(****************************** 10-001-0215-00-0 ************************************)
(*************************** ProBoxElement with one Motor *******************************)
// Configuration element 
fbEL_10_001_0215_00_0.ConfigElement.ElementName                     := '10-001-0215-00-0'; // Element name 
fbEL_10_001_0215_00_0.ConfigElement.eElementNumber                  := E_10_001_0215_00_0; // Number of the element 
fbEL_10_001_0215_00_0.ConfigElement.eSlaveElementNumber_34          := E_ElementNumber.E_BEGIN_ELEMENT; // Link from Master to slave element
fbEL_10_001_0215_00_0.ConfigElement.eElementType                    := E_ElementType.NO_TYPE; // No specific type

// Register element 
ElementRegistry[E_10_001_0215_00_0].Enable                          := TRUE; // Object is called
ElementRegistry[E_10_001_0215_00_0].eElementNumber                  := fbEL_10_001_0215_00_0.ConfigElement.eElementNumber; 

(****************************** 10-001-0215-01-0 ************************************)
(************************** ProBox Straight Transport *******************************)
// Configuration function
fbF_10_001_0215_01_0.ConfigFunction.FunctionName                       := '10-001-0215-01-0'; // Function name
fbF_10_001_0215_01_0.ConfigFunction.eFunctionNumber                    := F_10_001_0215_01_0; // Number of the function
fbF_10_001_0215_01_0.ConfigFunction.eElementLink                       := E_ElementNumber.E_10_001_0215_00_0;
fbF_10_001_0215_01_0.ConfigFunction.FunctionLink.eFunctionNumber       := E_FunctionNumber.F_BEGIN_FUNCTION;
fbF_10_001_0215_01_0.ConfigFunction.FunctionLink.ZoneNumber            := 0;
fbF_10_001_0215_01_0.ConfigFunction.eAdjacentFunctionNumberSide[1]     := E_FunctionNumber.F_10_001_0214_01_0;
fbF_10_001_0215_01_0.ConfigFunction.eAdjacentFunctionNumberSide[2]     := E_FunctionNumber.F_10_001_0215_02_0;
fbF_10_001_0215_01_0.ConfigFunction.ePrevFunctionNumber                := E_FunctionNumber.F_10_001_0214_01_0;
fbF_10_001_0215_01_0.ConfigFunction.eNextFunctionNumber                := E_FunctionNumber.F_10_001_0215_02_0;
fbF_10_001_0215_01_0.ConfigFunction.NumberOfZones                      := 1;
//Config zone 1
fbF_10_001_0215_01_0.ConfigFunction.Zone[1].ZoneName                   := '10-001-0215-01-1';
fbF_10_001_0215_01_0.ConfigFunction.Zone[1].EnableMFC                  := TRUE;
fbF_10_001_0215_01_0.ConfigFunction.Zone[1].EnableSimultaneousTransport:= FALSE; //Disable Simultaneous transport for multi zone functions
fbF_10_001_0215_01_0.ConfigFunction.Zone[1].EnableLatchOccupiedState   := TRUE;
fbF_10_001_0215_01_0.ConfigFunction.Zone[1].Length[1]                  := INT_TO_UINT(2600 / fbF_10_001_0215_01_0.ConfigFunction.NumberOfZones);	//Zone length (ie element length / number of zones)

// Register function
FunctionRegistry[F_10_001_0215_01_0].Enable                            := TRUE; (* Function will be called *)
FunctionRegistry[F_10_001_0215_01_0].eFunctionNumber                   := fbF_10_001_0215_01_0.ConfigFunction.eFunctionNumber; // Registration number


(****************************** 10-001-0215-02-0 ************************************)
(************************** ProBox Straight Transport *******************************)
// Configuration function
fbF_10_001_0215_02_0.ConfigFunction.FunctionName                       := '10-001-0215-02-0'; // Function name
fbF_10_001_0215_02_0.ConfigFunction.eFunctionNumber                    := F_10_001_0215_02_0; // Number of the function
fbF_10_001_0215_02_0.ConfigFunction.eElementLink                       := E_ElementNumber.E_10_001_0215_00_0;
fbF_10_001_0215_02_0.ConfigFunction.FunctionLink.eFunctionNumber       := E_FunctionNumber.F_BEGIN_FUNCTION;
fbF_10_001_0215_02_0.ConfigFunction.FunctionLink.ZoneNumber            := 0;
fbF_10_001_0215_02_0.ConfigFunction.eAdjacentFunctionNumberSide[1]     := E_FunctionNumber.F_10_001_0215_01_0;
fbF_10_001_0215_02_0.ConfigFunction.eAdjacentFunctionNumberSide[2]     := E_FunctionNumber.F_BEGIN_FUNCTION;
fbF_10_001_0215_02_0.ConfigFunction.ePrevFunctionNumber                := E_FunctionNumber.F_10_001_0215_01_0;
fbF_10_001_0215_02_0.ConfigFunction.eNextFunctionNumber                := E_FunctionNumber.F_BEGIN_FUNCTION;
fbF_10_001_0215_02_0.ConfigFunction.NumberOfZones                      := 1;
//Config zone 1
fbF_10_001_0215_02_0.ConfigFunction.Zone[1].ZoneName                   := '10-001-0215-02-1';
fbF_10_001_0215_02_0.ConfigFunction.Zone[1].EnableMFC                  := TRUE;
fbF_10_001_0215_02_0.ConfigFunction.Zone[1].EnableSimultaneousTransport:= FALSE; //Disable Simultaneous transport for multi zone functions
fbF_10_001_0215_02_0.ConfigFunction.Zone[1].EnableLatchOccupiedState   := TRUE;
fbF_10_001_0215_02_0.ConfigFunction.Zone[1].Length[1]                  := INT_TO_UINT(2600 / fbF_10_001_0215_02_0.ConfigFunction.NumberOfZones);	//Zone length (ie element length / number of zones)

// Register function
FunctionRegistry[F_10_001_0215_02_0].Enable                            := TRUE; (* Function will be called *)
FunctionRegistry[F_10_001_0215_02_0].eFunctionNumber                   := fbF_10_001_0215_02_0.ConfigFunction.eFunctionNumber; // Registration number


(****************************** 10-001-0215-03-0 ************************************)
(******************************* Crane Handover/Takeover ***********************************)
// Configuration function 
fbF_10_001_0215_03_0.ConfigFunction.FunctionName                      	 := '10-001-0215-03-0'; (* Function name *)
fbF_10_001_0215_03_0.ConfigFunction.eFunctionNumber                  	 := F_10_001_0215_03_0; (* Number of the function *)
fbF_10_001_0215_03_0.ConfigFunction.eElementLink                     	 := E_ElementNumber.E_10_001_0215_00_0; 
fbF_10_001_0215_03_0.ConfigFunction.FunctionLink.eFunctionNumber     	 := E_FunctionNumber.F_10_001_0215_01_0;	//Addon link to function, this is auto generated, an may need to be changed.
fbF_10_001_0215_03_0.ConfigFunction.FunctionLink.ZoneNumber         	 := 1;		

fbF_10_001_0215_03_0.Config.TimeoutValueLift							 := T#10S;								// Timeout value for lifting
fbF_10_001_0215_03_0.Config.HomePosFree								 := E_Positions_LiftControl.DOWN;		// Homeposition lift when zone free
fbF_10_001_0215_03_0.Config.HomePosOccupied							 := E_Positions_LiftControl.UP;			// Homeposition lift when zone occupied
fbF_10_001_0215_03_0.Config.CraneXoverType								 := E_CvCraneXoverType.eCOMBINATION; 	// Function Crane Deposit and Crane Pickup
fbF_10_001_0215_03_0.Config.LiftEnabled								 := FALSE;								// config if station has lift	
fbF_10_001_0215_03_0.Config.CfgMotorTransfer.EnableMotorTransferTU		 := FALSE;  								// Enable or Disable motor drive chain transfer 
fbF_10_001_0215_03_0.Config.CfgMotorTransfer.HandoverMotorDir			 := E_DriveDirection.FWD; 				// Direction during handover
fbF_10_001_0215_03_0.Config.CfgMotorTransfer.TakeoverMotorDir			 := E_DriveDirection.FWD; 				// Direction during takeover
fbF_10_001_0215_03_0.Config.CfgMotorTransfer.MotorDriveTimeout			 := T#20S;	
fbF_10_001_0215_03_0.Config.CfgMotorTransfer.MotorSpeed				 := E_ProBoxMotorSpeed.NORMAL;

fbF_10_001_0215_03_0.Config.CraneCom.TCP_IP_Config.ChannelName          := 'CraneTCPIPcom';
fbF_10_001_0215_03_0.Config.CraneCom.TCP_IP_Config.EnableConnection     := TRUE;
fbF_10_001_0215_03_0.Config.CraneCom.TCP_IP_Config.RemoteHost           := '192.168.1.1';
fbF_10_001_0215_03_0.Config.CraneCom.TCP_IP_Config.RemotePort           := 2011;
fbF_10_001_0215_03_0.Config.CraneCom.TCP_IP_Config.LocalHost            := '0.0.0.0';
fbF_10_001_0215_03_0.Config.CraneCom.TCP_IP_Config.LocalPort            := 5001;
fbF_10_001_0215_03_0.Config.CraneCom.TCP_IP_Config.Server               := FALSE;
fbF_10_001_0215_03_0.Config.CraneCom.TCP_IP_Config.ConnectTimeout       := T#10S;
fbF_10_001_0215_03_0.Config.CraneCom.TCP_IP_Config.ClientRetryInterval  := T#5S;
fbF_10_001_0215_03_0.Config.CraneCom.TCP_IP_Config.ServerRetryInterval  := T#1S;
fbF_10_001_0215_03_0.Config.CraneCom.TCP_IP_Config.AcceptPollInterval   := T#10S;
fbF_10_001_0215_03_0.Config.CraneCom.TCP_IP_Config.EnableDebugMsg       := TRUE;	


// Register function 
FunctionRegistry[F_10_001_0215_03_0].Enable                          	 := TRUE; (* Function will be called *)
FunctionRegistry[F_10_001_0215_03_0].eFunctionNumber                  	 := fbF_10_001_0215_03_0.ConfigFunction.eFunctionNumber; (* Registration number *)


(****************************** 10-001-0216-00-0 ************************************)
(*************************** ProBoxElement with one Motor *******************************)
// Configuration element 
fbEL_10_001_0216_00_0.ConfigElement.ElementName                     := '10-001-0216-00-0'; // Element name 
fbEL_10_001_0216_00_0.ConfigElement.eElementNumber                  := E_10_001_0216_00_0; // Number of the element 
fbEL_10_001_0216_00_0.ConfigElement.eSlaveElementNumber_34          := E_ElementNumber.E_BEGIN_ELEMENT; // Link from Master to slave element
fbEL_10_001_0216_00_0.ConfigElement.eElementType                    := E_ElementType.NO_TYPE; // No specific type

// Register element 
ElementRegistry[E_10_001_0216_00_0].Enable                          := TRUE; // Object is called
ElementRegistry[E_10_001_0216_00_0].eElementNumber                  := fbEL_10_001_0216_00_0.ConfigElement.eElementNumber; 

(****************************** 10-001-0216-01-0 ************************************)
(************************** ProBox Straight Transport *******************************)
// Configuration function
fbF_10_001_0216_01_0.ConfigFunction.FunctionName                       := '10-001-0216-01-0'; // Function name
fbF_10_001_0216_01_0.ConfigFunction.eFunctionNumber                    := F_10_001_0216_01_0; // Number of the function
fbF_10_001_0216_01_0.ConfigFunction.eElementLink                       := E_ElementNumber.E_10_001_0216_00_0;
fbF_10_001_0216_01_0.ConfigFunction.FunctionLink.eFunctionNumber       := E_FunctionNumber.F_BEGIN_FUNCTION;
fbF_10_001_0216_01_0.ConfigFunction.FunctionLink.ZoneNumber            := 0;
fbF_10_001_0216_01_0.ConfigFunction.eAdjacentFunctionNumberSide[1]     := E_FunctionNumber.F_BEGIN_FUNCTION;
fbF_10_001_0216_01_0.ConfigFunction.eAdjacentFunctionNumberSide[2]     := E_FunctionNumber.F_10_001_0217_01_0;
fbF_10_001_0216_01_0.ConfigFunction.ePrevFunctionNumber                := E_FunctionNumber.F_BEGIN_FUNCTION;
fbF_10_001_0216_01_0.ConfigFunction.eNextFunctionNumber                := E_FunctionNumber.F_10_001_0217_01_0;
fbF_10_001_0216_01_0.ConfigFunction.NumberOfZones                      := 2;
//Config zone 1
fbF_10_001_0216_01_0.ConfigFunction.Zone[1].ZoneName                   := '10-001-0216-01-1';
fbF_10_001_0216_01_0.ConfigFunction.Zone[1].EnableMFC                  := TRUE;
fbF_10_001_0216_01_0.ConfigFunction.Zone[1].EnableSimultaneousTransport:= TRUE; //Enable Simultaneous transport for multi zone functions
fbF_10_001_0216_01_0.ConfigFunction.Zone[1].EnableLatchOccupiedState   := TRUE;
fbF_10_001_0216_01_0.ConfigFunction.Zone[1].Length[1]                  := INT_TO_UINT(2600 / fbF_10_001_0216_01_0.ConfigFunction.NumberOfZones);	//Zone length (ie element length / number of zones)

//Config remaining zones equal to zone 1.
fbF_10_001_0216_01_0.ConfigFunction.Zone[2]                            := fbF_10_001_0216_01_0.ConfigFunction.Zone[1];
fbF_10_001_0216_01_0.ConfigFunction.Zone[2].ZoneName                   := '10-001-0216-01-2';

fbF_10_001_0216_01_0.Config.TwoSensorFunction                          := FALSE; // Slugging sensor present

// Register function
FunctionRegistry[F_10_001_0216_01_0].Enable                            := TRUE; (* Function will be called *)
FunctionRegistry[F_10_001_0216_01_0].eFunctionNumber                   := fbF_10_001_0216_01_0.ConfigFunction.eFunctionNumber; // Registration number


(****************************** 10-001-0216-02-0 ************************************)
(******************************* Crane Handover/Takeover ***********************************)
// Configuration function 
fbF_10_001_0216_02_0.ConfigFunction.FunctionName                      	 := '10-001-0216-02-0'; (* Function name *)
fbF_10_001_0216_02_0.ConfigFunction.eFunctionNumber                  	 := F_10_001_0216_02_0; (* Number of the function *)
fbF_10_001_0216_02_0.ConfigFunction.eElementLink                     	 := E_ElementNumber.E_10_001_0216_00_0; 
fbF_10_001_0216_02_0.ConfigFunction.FunctionLink.eFunctionNumber     	 := E_FunctionNumber.F_10_001_0216_01_0;	//Addon link to function, this is auto generated, an may need to be changed.
fbF_10_001_0216_02_0.ConfigFunction.FunctionLink.ZoneNumber         	 := 1;		

fbF_10_001_0216_02_0.Config.TimeoutValueLift							 := T#10S;								// Timeout value for lifting
fbF_10_001_0216_02_0.Config.HomePosFree								 := E_Positions_LiftControl.DOWN;		// Homeposition lift when zone free
fbF_10_001_0216_02_0.Config.HomePosOccupied							 := E_Positions_LiftControl.UP;			// Homeposition lift when zone occupied
fbF_10_001_0216_02_0.Config.CraneXoverType								 := E_CvCraneXoverType.eCOMBINATION; 	// Function Crane Deposit and Crane Pickup
fbF_10_001_0216_02_0.Config.LiftEnabled								 := FALSE;								// config if station has lift	
fbF_10_001_0216_02_0.Config.CfgMotorTransfer.EnableMotorTransferTU		 := FALSE;  								// Enable or Disable motor drive chain transfer 
fbF_10_001_0216_02_0.Config.CfgMotorTransfer.HandoverMotorDir			 := E_DriveDirection.FWD; 				// Direction during handover
fbF_10_001_0216_02_0.Config.CfgMotorTransfer.TakeoverMotorDir			 := E_DriveDirection.FWD; 				// Direction during takeover
fbF_10_001_0216_02_0.Config.CfgMotorTransfer.MotorDriveTimeout			 := T#20S;	
fbF_10_001_0216_02_0.Config.CfgMotorTransfer.MotorSpeed				 := E_ProBoxMotorSpeed.NORMAL;

fbF_10_001_0216_02_0.Config.CraneCom.TCP_IP_Config.ChannelName          := 'CraneTCPIPcom';
fbF_10_001_0216_02_0.Config.CraneCom.TCP_IP_Config.EnableConnection     := TRUE;
fbF_10_001_0216_02_0.Config.CraneCom.TCP_IP_Config.RemoteHost           := '192.168.1.1';
fbF_10_001_0216_02_0.Config.CraneCom.TCP_IP_Config.RemotePort           := 2011;
fbF_10_001_0216_02_0.Config.CraneCom.TCP_IP_Config.LocalHost            := '0.0.0.0';
fbF_10_001_0216_02_0.Config.CraneCom.TCP_IP_Config.LocalPort            := 5001;
fbF_10_001_0216_02_0.Config.CraneCom.TCP_IP_Config.Server               := FALSE;
fbF_10_001_0216_02_0.Config.CraneCom.TCP_IP_Config.ConnectTimeout       := T#10S;
fbF_10_001_0216_02_0.Config.CraneCom.TCP_IP_Config.ClientRetryInterval  := T#5S;
fbF_10_001_0216_02_0.Config.CraneCom.TCP_IP_Config.ServerRetryInterval  := T#1S;
fbF_10_001_0216_02_0.Config.CraneCom.TCP_IP_Config.AcceptPollInterval   := T#10S;
fbF_10_001_0216_02_0.Config.CraneCom.TCP_IP_Config.EnableDebugMsg       := TRUE;	


// Register function 
FunctionRegistry[F_10_001_0216_02_0].Enable                          	 := TRUE; (* Function will be called *)
FunctionRegistry[F_10_001_0216_02_0].eFunctionNumber                  	 := fbF_10_001_0216_02_0.ConfigFunction.eFunctionNumber; (* Registration number *)


(****************************** 10-001-0217-00-0 ************************************)
(*************************** ProBoxElement with one Motor *******************************)
// Configuration element 
fbEL_10_001_0217_00_0.ConfigElement.ElementName                     := '10-001-0217-00-0'; // Element name 
fbEL_10_001_0217_00_0.ConfigElement.eElementNumber                  := E_10_001_0217_00_0; // Number of the element 
fbEL_10_001_0217_00_0.ConfigElement.eSlaveElementNumber_34          := E_ElementNumber.E_BEGIN_ELEMENT; // Link from Master to slave element
fbEL_10_001_0217_00_0.ConfigElement.eElementType                    := E_ElementType.NO_TYPE; // No specific type

// Register element 
ElementRegistry[E_10_001_0217_00_0].Enable                          := TRUE; // Object is called
ElementRegistry[E_10_001_0217_00_0].eElementNumber                  := fbEL_10_001_0217_00_0.ConfigElement.eElementNumber; 

(****************************** 10-001-0217-01-0 ************************************)
(************************** ProBox Straight Transport *******************************)
// Configuration function
fbF_10_001_0217_01_0.ConfigFunction.FunctionName                       := '10-001-0217-01-0'; // Function name
fbF_10_001_0217_01_0.ConfigFunction.eFunctionNumber                    := F_10_001_0217_01_0; // Number of the function
fbF_10_001_0217_01_0.ConfigFunction.eElementLink                       := E_ElementNumber.E_10_001_0217_00_0;
fbF_10_001_0217_01_0.ConfigFunction.FunctionLink.eFunctionNumber       := E_FunctionNumber.F_BEGIN_FUNCTION;
fbF_10_001_0217_01_0.ConfigFunction.FunctionLink.ZoneNumber            := 0;
fbF_10_001_0217_01_0.ConfigFunction.eAdjacentFunctionNumberSide[1]     := E_FunctionNumber.F_10_001_0216_01_0;
fbF_10_001_0217_01_0.ConfigFunction.eAdjacentFunctionNumberSide[2]     := E_FunctionNumber.F_10_001_0212_01_0;
fbF_10_001_0217_01_0.ConfigFunction.ePrevFunctionNumber                := E_FunctionNumber.F_10_001_0216_01_0;
fbF_10_001_0217_01_0.ConfigFunction.eNextFunctionNumber                := E_FunctionNumber.F_10_001_0212_01_0;
fbF_10_001_0217_01_0.ConfigFunction.NumberOfZones                      := 1;
//Config zone 1
fbF_10_001_0217_01_0.ConfigFunction.Zone[1].ZoneName                   := '10-001-0217-01-1';
fbF_10_001_0217_01_0.ConfigFunction.Zone[1].EnableMFC                  := TRUE;
fbF_10_001_0217_01_0.ConfigFunction.Zone[1].EnableSimultaneousTransport:= FALSE; //Disable Simultaneous transport for multi zone functions
fbF_10_001_0217_01_0.ConfigFunction.Zone[1].EnableLatchOccupiedState   := TRUE;
fbF_10_001_0217_01_0.ConfigFunction.Zone[1].Length[1]                  := INT_TO_UINT(3000 / fbF_10_001_0217_01_0.ConfigFunction.NumberOfZones);	//Zone length (ie element length / number of zones)

// Register function
FunctionRegistry[F_10_001_0217_01_0].Enable                            := TRUE; (* Function will be called *)
FunctionRegistry[F_10_001_0217_01_0].eFunctionNumber                   := fbF_10_001_0217_01_0.ConfigFunction.eFunctionNumber; // Registration number


(****************************** 10-001-0218-00-0 ************************************)
(*************************** ProBoxElement with one Motor *******************************)
// Configuration element 
fbEL_10_001_0218_00_0.ConfigElement.ElementName                     := '10-001-0218-00-0'; // Element name 
fbEL_10_001_0218_00_0.ConfigElement.eElementNumber                  := E_10_001_0218_00_0; // Number of the element 
fbEL_10_001_0218_00_0.ConfigElement.eSlaveElementNumber_34          := E_ElementNumber.E_BEGIN_ELEMENT; // Link from Master to slave element
fbEL_10_001_0218_00_0.ConfigElement.eElementType                    := E_ElementType.NO_TYPE; // No specific type

// Register element 
ElementRegistry[E_10_001_0218_00_0].Enable                          := TRUE; // Object is called
ElementRegistry[E_10_001_0218_00_0].eElementNumber                  := fbEL_10_001_0218_00_0.ConfigElement.eElementNumber; 

(****************************** 10-001-0218-01-0 ************************************)
(************************** ProBox Straight Transport *******************************)
// Configuration function
fbF_10_001_0218_01_0.ConfigFunction.FunctionName                       := '10-001-0218-01-0'; // Function name
fbF_10_001_0218_01_0.ConfigFunction.eFunctionNumber                    := F_10_001_0218_01_0; // Number of the function
fbF_10_001_0218_01_0.ConfigFunction.eElementLink                       := E_ElementNumber.E_10_001_0218_00_0;
fbF_10_001_0218_01_0.ConfigFunction.FunctionLink.eFunctionNumber       := E_FunctionNumber.F_BEGIN_FUNCTION;
fbF_10_001_0218_01_0.ConfigFunction.FunctionLink.ZoneNumber            := 0;
fbF_10_001_0218_01_0.ConfigFunction.eAdjacentFunctionNumberSide[1]     := E_FunctionNumber.F_10_001_0212_01_0;
fbF_10_001_0218_01_0.ConfigFunction.eAdjacentFunctionNumberSide[2]     := E_FunctionNumber.F_10_001_0219_01_0;
fbF_10_001_0218_01_0.ConfigFunction.ePrevFunctionNumber                := E_FunctionNumber.F_10_001_0212_01_0;
fbF_10_001_0218_01_0.ConfigFunction.eNextFunctionNumber                := E_FunctionNumber.F_10_001_0219_01_0;
fbF_10_001_0218_01_0.ConfigFunction.NumberOfZones                      := 2;
//Config zone 1
fbF_10_001_0218_01_0.ConfigFunction.Zone[1].ZoneName                   := '10-001-0218-01-1';
fbF_10_001_0218_01_0.ConfigFunction.Zone[1].EnableMFC                  := TRUE;
fbF_10_001_0218_01_0.ConfigFunction.Zone[1].EnableSimultaneousTransport:= TRUE; //Enable Simultaneous transport for multi zone functions
fbF_10_001_0218_01_0.ConfigFunction.Zone[1].EnableLatchOccupiedState   := TRUE;
fbF_10_001_0218_01_0.ConfigFunction.Zone[1].Length[1]                  := INT_TO_UINT(2600 / fbF_10_001_0218_01_0.ConfigFunction.NumberOfZones);	//Zone length (ie element length / number of zones)

//Config remaining zones equal to zone 1.
fbF_10_001_0218_01_0.ConfigFunction.Zone[2]                            := fbF_10_001_0218_01_0.ConfigFunction.Zone[1];
fbF_10_001_0218_01_0.ConfigFunction.Zone[2].ZoneName                   := '10-001-0218-01-2';

fbF_10_001_0218_01_0.Config.TwoSensorFunction                          := FALSE; // Slugging sensor present

// Register function
FunctionRegistry[F_10_001_0218_01_0].Enable                            := TRUE; (* Function will be called *)
FunctionRegistry[F_10_001_0218_01_0].eFunctionNumber                   := fbF_10_001_0218_01_0.ConfigFunction.eFunctionNumber; // Registration number


(****************************** 10-001-0219-00-0 ************************************)
(*************************** ProBoxElement with one Motor *******************************)
// Configuration element 
fbEL_10_001_0219_00_0.ConfigElement.ElementName                     := '10-001-0219-00-0'; // Element name 
fbEL_10_001_0219_00_0.ConfigElement.eElementNumber                  := E_10_001_0219_00_0; // Number of the element 
fbEL_10_001_0219_00_0.ConfigElement.eSlaveElementNumber_34          := E_ElementNumber.E_BEGIN_ELEMENT; // Link from Master to slave element
fbEL_10_001_0219_00_0.ConfigElement.eElementType                    := E_ElementType.NO_TYPE; // No specific type

// Register element 
ElementRegistry[E_10_001_0219_00_0].Enable                          := TRUE; // Object is called
ElementRegistry[E_10_001_0219_00_0].eElementNumber                  := fbEL_10_001_0219_00_0.ConfigElement.eElementNumber; 

(****************************** 10-001-0219-01-0 ************************************)
(************************** ProBox Straight Transport *******************************)
// Configuration function
fbF_10_001_0219_01_0.ConfigFunction.FunctionName                       := '10-001-0219-01-0'; // Function name
fbF_10_001_0219_01_0.ConfigFunction.eFunctionNumber                    := F_10_001_0219_01_0; // Number of the function
fbF_10_001_0219_01_0.ConfigFunction.eElementLink                       := E_ElementNumber.E_10_001_0219_00_0;
fbF_10_001_0219_01_0.ConfigFunction.FunctionLink.eFunctionNumber       := E_FunctionNumber.F_BEGIN_FUNCTION;
fbF_10_001_0219_01_0.ConfigFunction.FunctionLink.ZoneNumber            := 0;
fbF_10_001_0219_01_0.ConfigFunction.eAdjacentFunctionNumberSide[1]     := E_FunctionNumber.F_10_001_0218_01_0;
fbF_10_001_0219_01_0.ConfigFunction.eAdjacentFunctionNumberSide[2]     := E_FunctionNumber.F_10_001_0220_01_0;
fbF_10_001_0219_01_0.ConfigFunction.ePrevFunctionNumber                := E_FunctionNumber.F_10_001_0218_01_0;
fbF_10_001_0219_01_0.ConfigFunction.eNextFunctionNumber                := E_FunctionNumber.F_10_001_0220_01_0;
fbF_10_001_0219_01_0.ConfigFunction.NumberOfZones                      := 2;
//Config zone 1
fbF_10_001_0219_01_0.ConfigFunction.Zone[1].ZoneName                   := '10-001-0219-01-1';
fbF_10_001_0219_01_0.ConfigFunction.Zone[1].EnableMFC                  := TRUE;
fbF_10_001_0219_01_0.ConfigFunction.Zone[1].EnableSimultaneousTransport:= TRUE; //Enable Simultaneous transport for multi zone functions
fbF_10_001_0219_01_0.ConfigFunction.Zone[1].EnableLatchOccupiedState   := TRUE;
fbF_10_001_0219_01_0.ConfigFunction.Zone[1].Length[1]                  := INT_TO_UINT(2600 / fbF_10_001_0219_01_0.ConfigFunction.NumberOfZones);	//Zone length (ie element length / number of zones)

//Config remaining zones equal to zone 1.
fbF_10_001_0219_01_0.ConfigFunction.Zone[2]                            := fbF_10_001_0219_01_0.ConfigFunction.Zone[1];
fbF_10_001_0219_01_0.ConfigFunction.Zone[2].ZoneName                   := '10-001-0219-01-2';

fbF_10_001_0219_01_0.Config.TwoSensorFunction                          := TRUE; // Slugging sensor present

// Register function
FunctionRegistry[F_10_001_0219_01_0].Enable                            := TRUE; (* Function will be called *)
FunctionRegistry[F_10_001_0219_01_0].eFunctionNumber                   := fbF_10_001_0219_01_0.ConfigFunction.eFunctionNumber; // Registration number


(****************************** 10-001-0220-00-0 ************************************)
(*************************** ProBoxElement with one Motor *******************************)
// Configuration element 
fbEL_10_001_0220_00_0.ConfigElement.ElementName                     := '10-001-0220-00-0'; // Element name 
fbEL_10_001_0220_00_0.ConfigElement.eElementNumber                  := E_10_001_0220_00_0; // Number of the element 
fbEL_10_001_0220_00_0.ConfigElement.eSlaveElementNumber_34          := E_ElementNumber.E_BEGIN_ELEMENT; // Link from Master to slave element
fbEL_10_001_0220_00_0.ConfigElement.eElementType                    := E_ElementType.NO_TYPE; // No specific type

// Register element 
ElementRegistry[E_10_001_0220_00_0].Enable                          := TRUE; // Object is called
ElementRegistry[E_10_001_0220_00_0].eElementNumber                  := fbEL_10_001_0220_00_0.ConfigElement.eElementNumber; 

(****************************** 10-001-0220-01-0 ************************************)
(************************** ProBox Straight Transport *******************************)
// Configuration function
fbF_10_001_0220_01_0.ConfigFunction.FunctionName                       := '10-001-0220-01-0'; // Function name
fbF_10_001_0220_01_0.ConfigFunction.eFunctionNumber                    := F_10_001_0220_01_0; // Number of the function
fbF_10_001_0220_01_0.ConfigFunction.eElementLink                       := E_ElementNumber.E_10_001_0220_00_0;
fbF_10_001_0220_01_0.ConfigFunction.FunctionLink.eFunctionNumber       := E_FunctionNumber.F_BEGIN_FUNCTION;
fbF_10_001_0220_01_0.ConfigFunction.FunctionLink.ZoneNumber            := 0;
fbF_10_001_0220_01_0.ConfigFunction.eAdjacentFunctionNumberSide[1]     := E_FunctionNumber.F_10_001_0219_01_0;
fbF_10_001_0220_01_0.ConfigFunction.eAdjacentFunctionNumberSide[2]     := E_FunctionNumber.F_10_001_0221_01_0;
fbF_10_001_0220_01_0.ConfigFunction.ePrevFunctionNumber                := E_FunctionNumber.F_10_001_0219_01_0;
fbF_10_001_0220_01_0.ConfigFunction.eNextFunctionNumber                := E_FunctionNumber.F_10_001_0221_01_0;
fbF_10_001_0220_01_0.ConfigFunction.NumberOfZones                      := 1;
//Config zone 1
fbF_10_001_0220_01_0.ConfigFunction.Zone[1].ZoneName                   := '10-001-0220-01-1';
fbF_10_001_0220_01_0.ConfigFunction.Zone[1].EnableMFC                  := TRUE;
fbF_10_001_0220_01_0.ConfigFunction.Zone[1].EnableSimultaneousTransport:= FALSE; //Disable Simultaneous transport for multi zone functions
fbF_10_001_0220_01_0.ConfigFunction.Zone[1].EnableLatchOccupiedState   := TRUE;
fbF_10_001_0220_01_0.ConfigFunction.Zone[1].Length[1]                  := INT_TO_UINT(3300 / fbF_10_001_0220_01_0.ConfigFunction.NumberOfZones);	//Zone length (ie element length / number of zones)

// Register function
FunctionRegistry[F_10_001_0220_01_0].Enable                            := TRUE; (* Function will be called *)
FunctionRegistry[F_10_001_0220_01_0].eFunctionNumber                   := fbF_10_001_0220_01_0.ConfigFunction.eFunctionNumber; // Registration number


(****************************** 10-001-0221-00-0 ************************************)
(*************************** ProBoxElement with one Motor *******************************)
// Configuration element 
fbEL_10_001_0221_00_0.ConfigElement.ElementName                     := '10-001-0221-00-0'; // Element name 
fbEL_10_001_0221_00_0.ConfigElement.eElementNumber                  := E_10_001_0221_00_0; // Number of the element 
fbEL_10_001_0221_00_0.ConfigElement.eSlaveElementNumber_34          := E_ElementNumber.E_10_001_0220_00_0; // Link from Master to slave element
fbEL_10_001_0221_00_0.ConfigElement.eElementType                    := E_ElementType.NO_TYPE; // No specific type

// Register element 
ElementRegistry[E_10_001_0221_00_0].Enable                          := TRUE; // Object is called
ElementRegistry[E_10_001_0221_00_0].eElementNumber                  := fbEL_10_001_0221_00_0.ConfigElement.eElementNumber; 

(****************************** 10-001-0221-01-0 ************************************)
(******************************** Transfer Unit *************************************)
// Configuration function
fbF_10_001_0221_01_0.ConfigFunction.FunctionName                    := '10-001-0221-01-0'; // Function name
fbF_10_001_0221_01_0.ConfigFunction.eFunctionNumber                 := F_10_001_0221_01_0; // Number of the function
fbF_10_001_0221_01_0.ConfigFunction.eElementLink                    := E_ElementNumber.E_10_001_0221_00_0;
fbF_10_001_0221_01_0.ConfigFunction.FunctionLink.eFunctionNumber    := E_FunctionNumber.F_BEGIN_FUNCTION;
fbF_10_001_0221_01_0.ConfigFunction.FunctionLink.ZoneNumber         := 0;
fbF_10_001_0221_01_0.ConfigFunction.eAdjacentFunctionNumberSide[1]  := E_FunctionNumber.F_BEGIN_FUNCTION;
fbF_10_001_0221_01_0.ConfigFunction.eAdjacentFunctionNumberSide[2]  := E_FunctionNumber.F_10_001_0222_01_0;
fbF_10_001_0221_01_0.ConfigFunction.eAdjacentFunctionNumberSide[3]  := E_FunctionNumber.F_10_001_0220_01_0;
fbF_10_001_0221_01_0.ConfigFunction.eAdjacentFunctionNumberSide[4]  := E_FunctionNumber.F_BEGIN_FUNCTION;
fbF_10_001_0221_01_0.ConfigFunction.ePrevFunctionNumber             := E_FunctionNumber.F_10_001_0220_01_0;
fbF_10_001_0221_01_0.ConfigFunction.eNextFunctionNumber             := E_FunctionNumber.F_10_001_0222_01_0;
fbF_10_001_0221_01_0.ConfigFunction.FlowDirectionREV                := FALSE;
fbF_10_001_0221_01_0.ConfigFunction.NumberOfZones                   := 1;

fbF_10_001_0221_01_0.ConfigFunction.Zone[1].ZoneName                := '10-001-0221-01-1';
fbF_10_001_0221_01_0.ConfigFunction.Zone[1].EnableMFC                 := TRUE;
fbF_10_001_0221_01_0.ConfigFunction.Zone[1].EnableLatchOccupiedState  := TRUE;
fbF_10_001_0221_01_0.ConfigFunction.Zone[1].Length[1]               := 1000;

fbF_10_001_0221_01_0.Config.TimeoutValueLift                        := T#15S; // Timeout value for lifting
fbF_10_001_0221_01_0.Config.HomePosFree                             := E_Positions_LiftControl.UNDIFINED; // Homeposition lift when zone free, UNDIFINED=> No home position is set, and lift stays where it is.
fbF_10_001_0221_01_0.Config.HomePosOccupied                         := E_Positions_LiftControl.UNDIFINED; // Homeposition lift when zone occupied, UNDIFINED=> No home position is set, and lift stays where it is.
fbF_10_001_0221_01_0.Config.LiftType                                := E_LiftType.E_LiftChain; // Configured lifting type, Roller or Chain
fbF_10_001_0221_01_0.Config.SingleTUMode							 := E_SingleTuMode.SingleTuMode; // Transfer unit and slave element's extended functions only allow one TU at a time. Change to optimize the transfer unit.

// Register function                                                     
FunctionRegistry[F_10_001_0221_01_0].Enable                         := TRUE; (* Function will be called *)
FunctionRegistry[F_10_001_0221_01_0].eFunctionNumber                := fbF_10_001_0221_01_0.ConfigFunction.eFunctionNumber; // Registration number


(****************************** 10-001-0222-00-0 ************************************)
(*************************** ProBoxElement with one Motor *******************************)
// Configuration element 
fbEL_10_001_0222_00_0.ConfigElement.ElementName                     := '10-001-0222-00-0'; // Element name 
fbEL_10_001_0222_00_0.ConfigElement.eElementNumber                  := E_10_001_0222_00_0; // Number of the element 
fbEL_10_001_0222_00_0.ConfigElement.eSlaveElementNumber_34          := E_ElementNumber.E_10_001_0223_00_0; // Link from Master to slave element
fbEL_10_001_0222_00_0.ConfigElement.eElementType                    := E_ElementType.NO_TYPE; // No specific type

// Register element 
ElementRegistry[E_10_001_0222_00_0].Enable                          := TRUE; // Object is called
ElementRegistry[E_10_001_0222_00_0].eElementNumber                  := fbEL_10_001_0222_00_0.ConfigElement.eElementNumber; 

(****************************** 10-001-0222-01-0 ************************************)
(******************************** Transfer Unit *************************************)
// Configuration function
fbF_10_001_0222_01_0.ConfigFunction.FunctionName                    := '10-001-0222-01-0'; // Function name
fbF_10_001_0222_01_0.ConfigFunction.eFunctionNumber                 := F_10_001_0222_01_0; // Number of the function
fbF_10_001_0222_01_0.ConfigFunction.eElementLink                    := E_ElementNumber.E_10_001_0222_00_0;
fbF_10_001_0222_01_0.ConfigFunction.FunctionLink.eFunctionNumber    := E_FunctionNumber.F_BEGIN_FUNCTION;
fbF_10_001_0222_01_0.ConfigFunction.FunctionLink.ZoneNumber         := 0;
fbF_10_001_0222_01_0.ConfigFunction.eAdjacentFunctionNumberSide[1]  := E_FunctionNumber.F_10_001_0221_01_0;
fbF_10_001_0222_01_0.ConfigFunction.eAdjacentFunctionNumberSide[2]  := E_FunctionNumber.F_10_001_0230_01_0;
fbF_10_001_0222_01_0.ConfigFunction.eAdjacentFunctionNumberSide[3]  := E_FunctionNumber.F_BEGIN_FUNCTION;
fbF_10_001_0222_01_0.ConfigFunction.eAdjacentFunctionNumberSide[4]  := E_FunctionNumber.F_10_001_0225_01_0;
fbF_10_001_0222_01_0.ConfigFunction.ePrevFunctionNumber             := E_FunctionNumber.F_10_001_0221_01_0;
fbF_10_001_0222_01_0.ConfigFunction.eNextFunctionNumber             := E_FunctionNumber.F_BEGIN_FUNCTION;
fbF_10_001_0222_01_0.ConfigFunction.FlowDirectionREV                := FALSE;
fbF_10_001_0222_01_0.ConfigFunction.NumberOfZones                   := 1;

fbF_10_001_0222_01_0.ConfigFunction.Zone[1].ZoneName                := '10-001-0222-01-1';
fbF_10_001_0222_01_0.ConfigFunction.Zone[1].EnableMFC                 := TRUE;
fbF_10_001_0222_01_0.ConfigFunction.Zone[1].EnableLatchOccupiedState  := TRUE;
fbF_10_001_0222_01_0.ConfigFunction.Zone[1].Length[1]               := 1000;

fbF_10_001_0222_01_0.Config.TimeoutValueLift                        := T#15S; // Timeout value for lifting
fbF_10_001_0222_01_0.Config.HomePosFree                             := E_Positions_LiftControl.UNDIFINED; // Homeposition lift when zone free, UNDIFINED=> No home position is set, and lift stays where it is.
fbF_10_001_0222_01_0.Config.HomePosOccupied                         := E_Positions_LiftControl.UNDIFINED; // Homeposition lift when zone occupied, UNDIFINED=> No home position is set, and lift stays where it is.
fbF_10_001_0222_01_0.Config.LiftType                                := E_LiftType.E_LiftChain; // Configured lifting type, Roller or Chain
fbF_10_001_0222_01_0.Config.SingleTUMode							 := E_SingleTuMode.SingleTuMode; // Transfer unit and slave element's extended functions only allow one TU at a time. Change to optimize the transfer unit.

// Register function                                                     
FunctionRegistry[F_10_001_0222_01_0].Enable                         := TRUE; (* Function will be called *)
FunctionRegistry[F_10_001_0222_01_0].eFunctionNumber                := fbF_10_001_0222_01_0.ConfigFunction.eFunctionNumber; // Registration number


(****************************** 10-001-0223-00-0 ************************************)
(*************************** ProBoxElement with one Motor *******************************)
// Configuration element 
fbEL_10_001_0223_00_0.ConfigElement.ElementName                     := '10-001-0223-00-0'; // Element name 
fbEL_10_001_0223_00_0.ConfigElement.eElementNumber                  := E_10_001_0223_00_0; // Number of the element 
fbEL_10_001_0223_00_0.ConfigElement.eSlaveElementNumber_34          := E_ElementNumber.E_BEGIN_ELEMENT; // Link from Master to slave element
fbEL_10_001_0223_00_0.ConfigElement.eElementType                    := E_ElementType.NO_TYPE; // No specific type

// Register element 
ElementRegistry[E_10_001_0223_00_0].Enable                          := TRUE; // Object is called
ElementRegistry[E_10_001_0223_00_0].eElementNumber                  := fbEL_10_001_0223_00_0.ConfigElement.eElementNumber; 

(****************************** 10-001-0225-00-0 ************************************)
(*************************** ProBoxElement with one Motor *******************************)
// Configuration element 
fbEL_10_001_0225_00_0.ConfigElement.ElementName                     := '10-001-0225-00-0'; // Element name 
fbEL_10_001_0225_00_0.ConfigElement.eElementNumber                  := E_10_001_0225_00_0; // Number of the element 
fbEL_10_001_0225_00_0.ConfigElement.eSlaveElementNumber_34          := E_ElementNumber.E_BEGIN_ELEMENT; // Link from Master to slave element
fbEL_10_001_0225_00_0.ConfigElement.eElementType                    := E_ElementType.NO_TYPE; // No specific type

// Register element 
ElementRegistry[E_10_001_0225_00_0].Enable                          := TRUE; // Object is called
ElementRegistry[E_10_001_0225_00_0].eElementNumber                  := fbEL_10_001_0225_00_0.ConfigElement.eElementNumber; 

(****************************** 10-001-0225-01-0 ************************************)
(************************** ProBox Straight Transport *******************************)
// Configuration function
fbF_10_001_0225_01_0.ConfigFunction.FunctionName                       := '10-001-0225-01-0'; // Function name
fbF_10_001_0225_01_0.ConfigFunction.eFunctionNumber                    := F_10_001_0225_01_0; // Number of the function
fbF_10_001_0225_01_0.ConfigFunction.eElementLink                       := E_ElementNumber.E_10_001_0225_00_0;
fbF_10_001_0225_01_0.ConfigFunction.FunctionLink.eFunctionNumber       := E_FunctionNumber.F_BEGIN_FUNCTION;
fbF_10_001_0225_01_0.ConfigFunction.FunctionLink.ZoneNumber            := 0;
fbF_10_001_0225_01_0.ConfigFunction.eAdjacentFunctionNumberSide[1]     := E_FunctionNumber.F_10_001_0222_01_0;
fbF_10_001_0225_01_0.ConfigFunction.eAdjacentFunctionNumberSide[2]     := E_FunctionNumber.F_10_001_0226_01_0;
fbF_10_001_0225_01_0.ConfigFunction.ePrevFunctionNumber                := E_FunctionNumber.F_10_001_0222_01_0;
fbF_10_001_0225_01_0.ConfigFunction.eNextFunctionNumber                := E_FunctionNumber.F_10_001_0226_01_0;
fbF_10_001_0225_01_0.ConfigFunction.NumberOfZones                      := 2;
//Config zone 1
fbF_10_001_0225_01_0.ConfigFunction.Zone[1].ZoneName                   := '10-001-0225-01-1';
fbF_10_001_0225_01_0.ConfigFunction.Zone[1].EnableMFC                  := TRUE;
fbF_10_001_0225_01_0.ConfigFunction.Zone[1].EnableSimultaneousTransport:= TRUE; //Enable Simultaneous transport for multi zone functions
fbF_10_001_0225_01_0.ConfigFunction.Zone[1].EnableLatchOccupiedState   := TRUE;
fbF_10_001_0225_01_0.ConfigFunction.Zone[1].Length[1]                  := INT_TO_UINT(2600 / fbF_10_001_0225_01_0.ConfigFunction.NumberOfZones);	//Zone length (ie element length / number of zones)

//Config remaining zones equal to zone 1.
fbF_10_001_0225_01_0.ConfigFunction.Zone[2]                            := fbF_10_001_0225_01_0.ConfigFunction.Zone[1];
fbF_10_001_0225_01_0.ConfigFunction.Zone[2].ZoneName                   := '10-001-0225-01-2';

fbF_10_001_0225_01_0.Config.TwoSensorFunction                          := FALSE; // Slugging sensor present

// Register function
FunctionRegistry[F_10_001_0225_01_0].Enable                            := TRUE; (* Function will be called *)
FunctionRegistry[F_10_001_0225_01_0].eFunctionNumber                   := fbF_10_001_0225_01_0.ConfigFunction.eFunctionNumber; // Registration number


(****************************** 10-001-0226-00-0 ************************************)
(*************************** ProBoxElement with one Motor *******************************)
// Configuration element 
fbEL_10_001_0226_00_0.ConfigElement.ElementName                     := '10-001-0226-00-0'; // Element name 
fbEL_10_001_0226_00_0.ConfigElement.eElementNumber                  := E_10_001_0226_00_0; // Number of the element 
fbEL_10_001_0226_00_0.ConfigElement.eSlaveElementNumber_34          := E_ElementNumber.E_BEGIN_ELEMENT; // Link from Master to slave element
fbEL_10_001_0226_00_0.ConfigElement.eElementType                    := E_ElementType.NO_TYPE; // No specific type

// Register element 
ElementRegistry[E_10_001_0226_00_0].Enable                          := TRUE; // Object is called
ElementRegistry[E_10_001_0226_00_0].eElementNumber                  := fbEL_10_001_0226_00_0.ConfigElement.eElementNumber; 

(****************************** 10-001-0226-01-0 ************************************)
(************************** ProBox Straight Transport *******************************)
// Configuration function
fbF_10_001_0226_01_0.ConfigFunction.FunctionName                       := '10-001-0226-01-0'; // Function name
fbF_10_001_0226_01_0.ConfigFunction.eFunctionNumber                    := F_10_001_0226_01_0; // Number of the function
fbF_10_001_0226_01_0.ConfigFunction.eElementLink                       := E_ElementNumber.E_10_001_0226_00_0;
fbF_10_001_0226_01_0.ConfigFunction.FunctionLink.eFunctionNumber       := E_FunctionNumber.F_BEGIN_FUNCTION;
fbF_10_001_0226_01_0.ConfigFunction.FunctionLink.ZoneNumber            := 0;
fbF_10_001_0226_01_0.ConfigFunction.eAdjacentFunctionNumberSide[1]     := E_FunctionNumber.F_10_001_0225_01_0;
fbF_10_001_0226_01_0.ConfigFunction.eAdjacentFunctionNumberSide[2]     := E_FunctionNumber.F_10_001_0227_01_0;
fbF_10_001_0226_01_0.ConfigFunction.ePrevFunctionNumber                := E_FunctionNumber.F_10_001_0225_01_0;
fbF_10_001_0226_01_0.ConfigFunction.eNextFunctionNumber                := E_FunctionNumber.F_10_001_0227_01_0;
fbF_10_001_0226_01_0.ConfigFunction.NumberOfZones                      := 2;
//Config zone 1
fbF_10_001_0226_01_0.ConfigFunction.Zone[1].ZoneName                   := '10-001-0226-01-1';
fbF_10_001_0226_01_0.ConfigFunction.Zone[1].EnableMFC                  := TRUE;
fbF_10_001_0226_01_0.ConfigFunction.Zone[1].EnableSimultaneousTransport:= TRUE; //Enable Simultaneous transport for multi zone functions
fbF_10_001_0226_01_0.ConfigFunction.Zone[1].EnableLatchOccupiedState   := TRUE;
fbF_10_001_0226_01_0.ConfigFunction.Zone[1].Length[1]                  := INT_TO_UINT(2600 / fbF_10_001_0226_01_0.ConfigFunction.NumberOfZones);	//Zone length (ie element length / number of zones)

//Config remaining zones equal to zone 1.
fbF_10_001_0226_01_0.ConfigFunction.Zone[2]                            := fbF_10_001_0226_01_0.ConfigFunction.Zone[1];
fbF_10_001_0226_01_0.ConfigFunction.Zone[2].ZoneName                   := '10-001-0226-01-2';

fbF_10_001_0226_01_0.Config.TwoSensorFunction                          := FALSE; // Slugging sensor present

// Register function
FunctionRegistry[F_10_001_0226_01_0].Enable                            := TRUE; (* Function will be called *)
FunctionRegistry[F_10_001_0226_01_0].eFunctionNumber                   := fbF_10_001_0226_01_0.ConfigFunction.eFunctionNumber; // Registration number


(****************************** 10-001-0227-00-0 ************************************)
(*************************** ProBoxElement with one Motor *******************************)
// Configuration element 
fbEL_10_001_0227_00_0.ConfigElement.ElementName                     := '10-001-0227-00-0'; // Element name 
fbEL_10_001_0227_00_0.ConfigElement.eElementNumber                  := E_10_001_0227_00_0; // Number of the element 
fbEL_10_001_0227_00_0.ConfigElement.eSlaveElementNumber_34          := E_ElementNumber.E_BEGIN_ELEMENT; // Link from Master to slave element
fbEL_10_001_0227_00_0.ConfigElement.eElementType                    := E_ElementType.NO_TYPE; // No specific type

// Register element 
ElementRegistry[E_10_001_0227_00_0].Enable                          := TRUE; // Object is called
ElementRegistry[E_10_001_0227_00_0].eElementNumber                  := fbEL_10_001_0227_00_0.ConfigElement.eElementNumber; 

(****************************** 10-001-0227-01-0 ************************************)
(************************** ProBox Straight Transport *******************************)
// Configuration function
fbF_10_001_0227_01_0.ConfigFunction.FunctionName                       := '10-001-0227-01-0'; // Function name
fbF_10_001_0227_01_0.ConfigFunction.eFunctionNumber                    := F_10_001_0227_01_0; // Number of the function
fbF_10_001_0227_01_0.ConfigFunction.eElementLink                       := E_ElementNumber.E_10_001_0227_00_0;
fbF_10_001_0227_01_0.ConfigFunction.FunctionLink.eFunctionNumber       := E_FunctionNumber.F_BEGIN_FUNCTION;
fbF_10_001_0227_01_0.ConfigFunction.FunctionLink.ZoneNumber            := 0;
fbF_10_001_0227_01_0.ConfigFunction.eAdjacentFunctionNumberSide[1]     := E_FunctionNumber.F_10_001_0226_01_0;
fbF_10_001_0227_01_0.ConfigFunction.eAdjacentFunctionNumberSide[2]     := E_FunctionNumber.F_10_001_0209_01_0;
fbF_10_001_0227_01_0.ConfigFunction.ePrevFunctionNumber                := E_FunctionNumber.F_10_001_0226_01_0;
fbF_10_001_0227_01_0.ConfigFunction.eNextFunctionNumber                := E_FunctionNumber.F_10_001_0209_01_0;
fbF_10_001_0227_01_0.ConfigFunction.NumberOfZones                      := 1;
//Config zone 1
fbF_10_001_0227_01_0.ConfigFunction.Zone[1].ZoneName                   := '10-001-0227-01-1';
fbF_10_001_0227_01_0.ConfigFunction.Zone[1].EnableMFC                  := TRUE;
fbF_10_001_0227_01_0.ConfigFunction.Zone[1].EnableSimultaneousTransport:= FALSE; //Disable Simultaneous transport for multi zone functions
fbF_10_001_0227_01_0.ConfigFunction.Zone[1].EnableLatchOccupiedState   := TRUE;
fbF_10_001_0227_01_0.ConfigFunction.Zone[1].Length[1]                  := INT_TO_UINT(1400 / fbF_10_001_0227_01_0.ConfigFunction.NumberOfZones);	//Zone length (ie element length / number of zones)

// Register function
FunctionRegistry[F_10_001_0227_01_0].Enable                            := TRUE; (* Function will be called *)
FunctionRegistry[F_10_001_0227_01_0].eFunctionNumber                   := fbF_10_001_0227_01_0.ConfigFunction.eFunctionNumber; // Registration number


(****************************** 10-001-0230-00-0 ************************************)
(*************************** ProBoxElement with one Motor *******************************)
// Configuration element 
fbEL_10_001_0230_00_0.ConfigElement.ElementName                     := '10-001-0230-00-0'; // Element name 
fbEL_10_001_0230_00_0.ConfigElement.eElementNumber                  := E_10_001_0230_00_0; // Number of the element 
fbEL_10_001_0230_00_0.ConfigElement.eSlaveElementNumber_34          := E_ElementNumber.E_BEGIN_ELEMENT; // Link from Master to slave element
fbEL_10_001_0230_00_0.ConfigElement.eElementType                    := E_ElementType.NO_TYPE; // No specific type

// Register element 
ElementRegistry[E_10_001_0230_00_0].Enable                          := TRUE; // Object is called
ElementRegistry[E_10_001_0230_00_0].eElementNumber                  := fbEL_10_001_0230_00_0.ConfigElement.eElementNumber; 

(****************************** 10-001-0230-01-0 ************************************)
(******************************** TransferCC  ***************************************)
// Configuration function
fbF_10_001_0230_01_0.ConfigFunction.FunctionName                      := '10-001-0230-01-0'; // Function name
fbF_10_001_0230_01_0.ConfigFunction.eFunctionNumber                   := F_10_001_0230_01_0; // Number of the function
fbF_10_001_0230_01_0.ConfigFunction.eElementLink                      := E_ElementNumber.E_10_001_0230_00_0;
fbF_10_001_0230_01_0.ConfigFunction.FunctionLink.eFunctionNumber      := E_FunctionNumber.F_BEGIN_FUNCTION;
fbF_10_001_0230_01_0.ConfigFunction.FunctionLink.ZoneNumber           := 0;
fbF_10_001_0230_01_0.ConfigFunction.eAdjacentFunctionNumberSide[1]    := E_FunctionNumber.F_10_001_0222_01_0;
fbF_10_001_0230_01_0.ConfigFunction.eAdjacentFunctionNumberSide[2]    := E_FunctionNumber.F_10_001_0232_01_0;
fbF_10_001_0230_01_0.ConfigFunction.eAdjacentFunctionNumberSide[3]    := E_FunctionNumber.F_BEGIN_FUNCTION;
fbF_10_001_0230_01_0.ConfigFunction.eAdjacentFunctionNumberSide[4]    := E_FunctionNumber.F_BEGIN_FUNCTION;
fbF_10_001_0230_01_0.ConfigFunction.ePrevFunctionNumber               := E_FunctionNumber.F_10_001_0222_01_0;
fbF_10_001_0230_01_0.ConfigFunction.eNextFunctionNumber               := E_FunctionNumber.F_10_001_0232_01_0;
fbF_10_001_0230_01_0.ConfigFunction.FlowDirectionREV                  := FALSE;
fbF_10_001_0230_01_0.ConfigFunction.NumberOfZones                     := 1;

fbF_10_001_0230_01_0.ConfigFunction.Zone[1].ZoneName                  := '10-001-0230-01-1';
fbF_10_001_0230_01_0.ConfigFunction.Zone[1].EnableMFC                 := TRUE;
fbF_10_001_0230_01_0.ConfigFunction.Zone[1].EnableLatchOccupiedState  := TRUE;
fbF_10_001_0230_01_0.ConfigFunction.Zone[1].Length[1]                 := 1400;


fbF_10_001_0230_01_0.Config.HomePosFree								  := E_Positions_HorizontalControl.LEFT;
fbF_10_001_0230_01_0.Config.HomePosOccupied							  := E_Positions_HorizontalControl.LEFT;
fbF_10_001_0230_01_0.Config.ReleaseBreakTime						  := T#500MS;
fbF_10_001_0230_01_0.Config.TimeoutValueMotor						  := T#30S;

// Register function
FunctionRegistry[F_10_001_0230_01_0].Enable                     		:= TRUE; (* Function will be called *)
FunctionRegistry[F_10_001_0230_01_0].eFunctionNumber 					:= fbF_10_001_0230_01_0.ConfigFunction.eFunctionNumber; // Registration number


(****************************** 10-001-0232-00-0 ************************************)
(*************************** ProBoxElement with one Motor *******************************)
// Configuration element 
fbEL_10_001_0232_00_0.ConfigElement.ElementName                     := '10-001-0232-00-0'; // Element name 
fbEL_10_001_0232_00_0.ConfigElement.eElementNumber                  := E_10_001_0232_00_0; // Number of the element 
fbEL_10_001_0232_00_0.ConfigElement.eSlaveElementNumber_34          := E_ElementNumber.E_BEGIN_ELEMENT; // Link from Master to slave element
fbEL_10_001_0232_00_0.ConfigElement.eElementType                    := E_ElementType.NO_TYPE; // No specific type

// Register element 
ElementRegistry[E_10_001_0232_00_0].Enable                          := TRUE; // Object is called
ElementRegistry[E_10_001_0232_00_0].eElementNumber                  := fbEL_10_001_0232_00_0.ConfigElement.eElementNumber; 

(****************************** 10-001-0232-01-0 ************************************)
(************************** ProBox Straight Transport *******************************)
// Configuration function
fbF_10_001_0232_01_0.ConfigFunction.FunctionName                       := '10-001-0232-01-0'; // Function name
fbF_10_001_0232_01_0.ConfigFunction.eFunctionNumber                    := F_10_001_0232_01_0; // Number of the function
fbF_10_001_0232_01_0.ConfigFunction.eElementLink                       := E_ElementNumber.E_10_001_0232_00_0;
fbF_10_001_0232_01_0.ConfigFunction.FunctionLink.eFunctionNumber       := E_FunctionNumber.F_BEGIN_FUNCTION;
fbF_10_001_0232_01_0.ConfigFunction.FunctionLink.ZoneNumber            := 0;
fbF_10_001_0232_01_0.ConfigFunction.eAdjacentFunctionNumberSide[1]     := E_FunctionNumber.F_10_001_0230_01_0;
fbF_10_001_0232_01_0.ConfigFunction.eAdjacentFunctionNumberSide[2]     := E_FunctionNumber.F_BEGIN_FUNCTION;
fbF_10_001_0232_01_0.ConfigFunction.ePrevFunctionNumber                := E_FunctionNumber.F_10_001_0230_01_0;
fbF_10_001_0232_01_0.ConfigFunction.eNextFunctionNumber                := E_FunctionNumber.F_BEGIN_FUNCTION;
fbF_10_001_0232_01_0.ConfigFunction.NumberOfZones                      := 2;
//Config zone 1
fbF_10_001_0232_01_0.ConfigFunction.Zone[1].ZoneName                   := '10-001-0232-01-1';
fbF_10_001_0232_01_0.ConfigFunction.Zone[1].EnableMFC                  := TRUE;
fbF_10_001_0232_01_0.ConfigFunction.Zone[1].EnableSimultaneousTransport:= TRUE; //Enable Simultaneous transport for multi zone functions
fbF_10_001_0232_01_0.ConfigFunction.Zone[1].EnableLatchOccupiedState   := TRUE;
fbF_10_001_0232_01_0.ConfigFunction.Zone[1].Length[1]                  := INT_TO_UINT(3000 / fbF_10_001_0232_01_0.ConfigFunction.NumberOfZones);	//Zone length (ie element length / number of zones)

//Config remaining zones equal to zone 1.
fbF_10_001_0232_01_0.ConfigFunction.Zone[2]                            := fbF_10_001_0232_01_0.ConfigFunction.Zone[1];
fbF_10_001_0232_01_0.ConfigFunction.Zone[2].ZoneName                   := '10-001-0232-01-2';

fbF_10_001_0232_01_0.Config.TwoSensorFunction                          := TRUE; // Slugging sensor present

// Register function
FunctionRegistry[F_10_001_0232_01_0].Enable                            := TRUE; (* Function will be called *)
FunctionRegistry[F_10_001_0232_01_0].eFunctionNumber                   := fbF_10_001_0232_01_0.ConfigFunction.eFunctionNumber; // Registration number


(****************************** 10-001-0232-02-0 ************************************)
(********************************* In/Out Feed ****************************************)
// Configuration function 
fbF_10_001_0232_02_0.ConfigFunction.FunctionName                     := '10-001-0232-02-0'; (* Function name *)
fbF_10_001_0232_02_0.ConfigFunction.eFunctionNumber                  := F_10_001_0232_02_0; (* Number of the function *)
fbF_10_001_0232_02_0.ConfigFunction.eElementLink                     := E_ElementNumber.E_10_001_0232_00_0; 
fbF_10_001_0232_02_0.ConfigFunction.FunctionLink.eFunctionNumber     := E_FunctionNumber.F_10_001_0232_01_0;	//Addon link to function, this is auto generated, an may need to be changed.
fbF_10_001_0232_02_0.ConfigFunction.FunctionLink.ZoneNumber          := 1;		

fbF_10_001_0232_02_0.Config.tFTLClearTime                  		  := T#5S; //Fork Truck Lift clear time
fbF_10_001_0232_02_0.Config.tTUSensorTime					  		  := T#5S; //Sensor occupied Time when to add or remove TU
fbF_10_001_0232_02_0.Config.TimeoutValueLift					  	  := T#10S; //Timeout value for lifting
fbF_10_001_0232_02_0.Config.LiftEnabled					  	  	  := FALSE; //Config if function has lift

// Register function 
FunctionRegistry[F_10_001_0232_02_0].Enable                           := TRUE; (* Function will be called *)
FunctionRegistry[F_10_001_0232_02_0].eFunctionNumber                  := fbF_10_001_0232_02_0.ConfigFunction.eFunctionNumber; (* Registration number *)


(****************************** 10-001-0233-00-0 ************************************)
(*************************** ProBoxElement with one Motor *******************************)
// Configuration element 
fbEL_10_001_0233_00_0.ConfigElement.ElementName                     := '10-001-0233-00-0'; // Element name 
fbEL_10_001_0233_00_0.ConfigElement.eElementNumber                  := E_10_001_0233_00_0; // Number of the element 
fbEL_10_001_0233_00_0.ConfigElement.eSlaveElementNumber_34          := E_ElementNumber.E_BEGIN_ELEMENT; // Link from Master to slave element
fbEL_10_001_0233_00_0.ConfigElement.eElementType                    := E_ElementType.NO_TYPE; // No specific type

// Register element 
ElementRegistry[E_10_001_0233_00_0].Enable                          := TRUE; // Object is called
ElementRegistry[E_10_001_0233_00_0].eElementNumber                  := fbEL_10_001_0233_00_0.ConfigElement.eElementNumber; 

(****************************** 10-001-0233-01-0 ************************************)
(************************** ProBox Straight Transport *******************************)
// Configuration function
fbF_10_001_0233_01_0.ConfigFunction.FunctionName                       := '10-001-0233-01-0'; // Function name
fbF_10_001_0233_01_0.ConfigFunction.eFunctionNumber                    := F_10_001_0233_01_0; // Number of the function
fbF_10_001_0233_01_0.ConfigFunction.eElementLink                       := E_ElementNumber.E_10_001_0233_00_0;
fbF_10_001_0233_01_0.ConfigFunction.FunctionLink.eFunctionNumber       := E_FunctionNumber.F_BEGIN_FUNCTION;
fbF_10_001_0233_01_0.ConfigFunction.FunctionLink.ZoneNumber            := 0;
fbF_10_001_0233_01_0.ConfigFunction.eAdjacentFunctionNumberSide[1]     := E_FunctionNumber.F_10_001_0204_01_0;
fbF_10_001_0233_01_0.ConfigFunction.eAdjacentFunctionNumberSide[2]     := E_FunctionNumber.F_BEGIN_FUNCTION;
fbF_10_001_0233_01_0.ConfigFunction.ePrevFunctionNumber                := E_FunctionNumber.F_10_001_0204_01_0;
fbF_10_001_0233_01_0.ConfigFunction.eNextFunctionNumber                := E_FunctionNumber.F_BEGIN_FUNCTION;
fbF_10_001_0233_01_0.ConfigFunction.NumberOfZones                      := 1;
//Config zone 1
fbF_10_001_0233_01_0.ConfigFunction.Zone[1].ZoneName                   := '10-001-0233-01-1';
fbF_10_001_0233_01_0.ConfigFunction.Zone[1].EnableMFC                  := TRUE;
fbF_10_001_0233_01_0.ConfigFunction.Zone[1].EnableSimultaneousTransport:= FALSE; //Disable Simultaneous transport for multi zone functions
fbF_10_001_0233_01_0.ConfigFunction.Zone[1].EnableLatchOccupiedState   := TRUE;
fbF_10_001_0233_01_0.ConfigFunction.Zone[1].Length[1]                  := INT_TO_UINT(1600 / fbF_10_001_0233_01_0.ConfigFunction.NumberOfZones);	//Zone length (ie element length / number of zones)

// Register function
FunctionRegistry[F_10_001_0233_01_0].Enable                            := TRUE; (* Function will be called *)
FunctionRegistry[F_10_001_0233_01_0].eFunctionNumber                   := fbF_10_001_0233_01_0.ConfigFunction.eFunctionNumber; // Registration number

END_FUNCTION

// ---- 10_Project/10_App/10_Config/F_ConfigPosition_002.TcPOU
FUNCTION F_ConfigPosition_002



(****************************** 10-002-0206-00-0 ************************************)
(*************************** ProBoxElement with one Motor *******************************)
// Configuration element 
fbEL_10_002_0206_00_0.ConfigElement.ElementName                     := '10-002-0206-00-0'; // Element name 
fbEL_10_002_0206_00_0.ConfigElement.eElementNumber                  := E_10_002_0206_00_0; // Number of the element 
fbEL_10_002_0206_00_0.ConfigElement.eSlaveElementNumber_34          := E_ElementNumber.E_BEGIN_ELEMENT; // Link from Master to slave element
fbEL_10_002_0206_00_0.ConfigElement.eElementType                    := E_ElementType.NO_TYPE; // No specific type

// Register element 
ElementRegistry[E_10_002_0206_00_0].Enable                          := TRUE; // Object is called
ElementRegistry[E_10_002_0206_00_0].eElementNumber                  := fbEL_10_002_0206_00_0.ConfigElement.eElementNumber; 

(****************************** 10-002-0206-01-0 ************************************)
(************************** ProBox Straight Transport *******************************)
// Configuration function
fbF_10_002_0206_01_0.ConfigFunction.FunctionName                       := '10-002-0206-01-0'; // Function name
fbF_10_002_0206_01_0.ConfigFunction.eFunctionNumber                    := F_10_002_0206_01_0; // Number of the function
fbF_10_002_0206_01_0.ConfigFunction.eElementLink                       := E_ElementNumber.E_10_002_0206_00_0;
fbF_10_002_0206_01_0.ConfigFunction.FunctionLink.eFunctionNumber       := E_FunctionNumber.F_BEGIN_FUNCTION;
fbF_10_002_0206_01_0.ConfigFunction.FunctionLink.ZoneNumber            := 0;
fbF_10_002_0206_01_0.ConfigFunction.eAdjacentFunctionNumberSide[1]     := E_FunctionNumber.F_10_001_0204_01_0;
fbF_10_002_0206_01_0.ConfigFunction.eAdjacentFunctionNumberSide[2]     := E_FunctionNumber.F_10_001_0208_01_0;
fbF_10_002_0206_01_0.ConfigFunction.ePrevFunctionNumber                := E_FunctionNumber.F_10_001_0204_01_0;
fbF_10_002_0206_01_0.ConfigFunction.eNextFunctionNumber                := E_FunctionNumber.F_10_001_0208_01_0;
fbF_10_002_0206_01_0.ConfigFunction.NumberOfZones                      := 1;
//Config zone 1
fbF_10_002_0206_01_0.ConfigFunction.Zone[1].ZoneName                   := '10-002-0206-01-1';
fbF_10_002_0206_01_0.ConfigFunction.Zone[1].EnableMFC                  := TRUE;
fbF_10_002_0206_01_0.ConfigFunction.Zone[1].EnableSimultaneousTransport:= FALSE; //Disable Simultaneous transport for multi zone functions
fbF_10_002_0206_01_0.ConfigFunction.Zone[1].EnableLatchOccupiedState   := TRUE;
fbF_10_002_0206_01_0.ConfigFunction.Zone[1].Length[1]                  := INT_TO_UINT(3000 / fbF_10_002_0206_01_0.ConfigFunction.NumberOfZones);	//Zone length (ie element length / number of zones)

// Register function
FunctionRegistry[F_10_002_0206_01_0].Enable                            := TRUE; (* Function will be called *)
FunctionRegistry[F_10_002_0206_01_0].eFunctionNumber                   := fbF_10_002_0206_01_0.ConfigFunction.eFunctionNumber; // Registration number

END_FUNCTION

// ---- 10_Project/10_App/10_Config/F_ConfigGroup.TcPOU
FUNCTION F_ConfigGroup



(********************************* Group 001 *************************************
 Switching Group 001 
**********************************************************************************)

fbSG_001.ConfigGroup.GroupName           			:= '10-001-0000-00-0'; 
fbSG_001.ConfigGroup.eGroupNumber         			:= E_GroupNumber.G_SG_001; 
fbSG_001.ConfigGroup.eGroupType                    := E_GroupType.SG;

fbSG_001.Config.NumberOfContactors                 := 8;
fbSG_001.Config.NumberOfAPs						:= 0;
fbSG_001.Config.AutoResetEmergencyCircuit          := FALSE;
fbSG_001.Config.ResetMemberElements                := TRUE;
fbSG_001.Config.tForcedStopDelay					:= T#30S;
fbSG_001.Config.tStartupDelay						:= T#5S;
fbSG_001.Config.tResetPulse                        := T#10ms;
fbSG_001.Config.FireAlarmUsed                      := TRUE;

GroupRegistry[E_GroupNumber.G_SG_001].Enable		:= TRUE;
GroupRegistry[E_GroupNumber.G_SG_001].eGroupNumber	:= fbSG_001.ConfigGroup.eGroupNumber;

(********************************* Group 002 *************************************
 Switching Group 002 
**********************************************************************************)

fbSG_002.ConfigGroup.GroupName           			:= '10-002-0000-00-0'; 
fbSG_002.ConfigGroup.eGroupNumber         			:= E_GroupNumber.G_SG_002; 
fbSG_002.ConfigGroup.eGroupType                    := E_GroupType.SG;

fbSG_002.Config.NumberOfContactors                 := 8;
fbSG_002.Config.NumberOfAPs						:= 0;
fbSG_002.Config.AutoResetEmergencyCircuit          := FALSE;
fbSG_002.Config.ResetMemberElements                := TRUE;
fbSG_002.Config.tForcedStopDelay					:= T#30S;
fbSG_002.Config.tStartupDelay						:= T#5S;
fbSG_002.Config.tResetPulse                        := T#10ms;
fbSG_002.Config.FireAlarmUsed                      := TRUE;

GroupRegistry[E_GroupNumber.G_SG_002].Enable		:= TRUE;
GroupRegistry[E_GroupNumber.G_SG_002].eGroupNumber	:= fbSG_002.ConfigGroup.eGroupNumber;

END_FUNCTION

// ---- 10_Project/10_App/10_Config/F_ConfigGroupManager.TcPOU
FUNCTION F_ConfigGroupManager



fbGroupManager.Config.Group[G_SG_001].eMemberElement[1]     := E_10_001_0200_00_0;
fbGroupManager.Config.Group[G_SG_001].eMemberElement[2]     := E_10_001_0201_00_0;
fbGroupManager.Config.Group[G_SG_001].eMemberElement[3]     := E_10_001_0202_00_0;
fbGroupManager.Config.Group[G_SG_001].eMemberElement[4]     := E_10_001_0203_00_0;
fbGroupManager.Config.Group[G_SG_001].eMemberElement[5]     := E_10_001_0204_00_0;
fbGroupManager.Config.Group[G_SG_001].eMemberElement[6]     := E_10_001_0205_00_0;
fbGroupManager.Config.Group[G_SG_001].eMemberElement[7]     := E_10_001_0207_00_0;
fbGroupManager.Config.Group[G_SG_001].eMemberElement[8]     := E_10_001_0208_00_0;
fbGroupManager.Config.Group[G_SG_001].eMemberElement[9]     := E_10_001_0209_00_0;
fbGroupManager.Config.Group[G_SG_001].eMemberElement[10]     := E_10_001_0211_00_0;
fbGroupManager.Config.Group[G_SG_001].eMemberElement[11]     := E_10_001_0212_00_0;
fbGroupManager.Config.Group[G_SG_001].eMemberElement[12]     := E_10_001_0213_00_0;
fbGroupManager.Config.Group[G_SG_001].eMemberElement[13]     := E_10_001_0214_00_0;
fbGroupManager.Config.Group[G_SG_001].eMemberElement[14]     := E_10_001_0215_00_0;
fbGroupManager.Config.Group[G_SG_001].eMemberElement[15]     := E_10_001_0216_00_0;
fbGroupManager.Config.Group[G_SG_001].eMemberElement[16]     := E_10_001_0217_00_0;
fbGroupManager.Config.Group[G_SG_001].eMemberElement[17]     := E_10_001_0218_00_0;
fbGroupManager.Config.Group[G_SG_001].eMemberElement[18]     := E_10_001_0219_00_0;
fbGroupManager.Config.Group[G_SG_001].eMemberElement[19]     := E_10_001_0220_00_0;
fbGroupManager.Config.Group[G_SG_001].eMemberElement[20]     := E_10_001_0221_00_0;
fbGroupManager.Config.Group[G_SG_001].eMemberElement[21]     := E_10_001_0222_00_0;
fbGroupManager.Config.Group[G_SG_001].eMemberElement[22]     := E_10_001_0223_00_0;
fbGroupManager.Config.Group[G_SG_001].eMemberElement[23]     := E_10_001_0225_00_0;
fbGroupManager.Config.Group[G_SG_001].eMemberElement[24]     := E_10_001_0226_00_0;
fbGroupManager.Config.Group[G_SG_001].eMemberElement[25]     := E_10_001_0227_00_0;
fbGroupManager.Config.Group[G_SG_001].eMemberElement[26]     := E_10_001_0230_00_0;
fbGroupManager.Config.Group[G_SG_001].eMemberElement[27]     := E_10_001_0232_00_0;
fbGroupManager.Config.Group[G_SG_001].eMemberElement[28]     := E_10_001_0233_00_0;
fbGroupManager.Config.Group[G_SG_002].eMemberElement[1]     := E_10_002_0206_00_0;

END_FUNCTION

// ---- 10_Project/10_App/10_Config/F_ConfigSubSystem.TcPOU
FUNCTION F_ConfigSubSystem : BOOL


(***********************************************************************************
   Subsystem 10
 ***********************************************************************************)
fbSubsystem10.ConfigSubsystem.SubSystemName         := '10-000-0000-000';
fbSubsystem10.ConfigSubsystem.SubsystemNumber       := 10;
fbSubsystem10.ConfigSubsystem.MaxMasterSpeed        := 100;
fbSubsystem10.ConfigSubsystem.MinMasterSpeed        := 50;
fbSubsystem10.ConfigSubsystem.MaxInitCallsPerCycle  := 10;
fbSubsystem10.Config.CPU_FanExists                  := FALSE;
fbSubsystem10.Config.MinFanSpeed                    := 0;
fbSubsystem10.Config.AM_Exists                      := TRUE;
fbSubsystem10.Config.SPOC_Exists                    := TRUE;
fbSubsystem10.Config.tDelayMonitoring               := T#2S;
fbSubsystem10.Config.tDelayStopping                 := T#1M;
fbSubsystem10.Config.EnableTimeSync                 := TRUE;
fbSubsystem10.Config.MinTimeSync                    := T#24H;
fbSubsystem10.Config.tRequestReset                  := T#1M;
fbSubsystem10.Config.CPU_UsageWarning               := 50;
fbSubsystem10.Config.CPU_UsageError                 := 60;
fbSubsystem10.Config.CPU_TemperatureWarning         := 85;
fbSubsystem10.Config.CPU_TemperatureError           := 95;

END_FUNCTION

// ---- 10_Project/10_App/10_Config/F_ConfigExternalDestination.TcPOU
FUNCTION F_ConfigExternalDestination : BOOL



;

END_FUNCTION

// ---- 20_Product/10_BCF/10_Base/11_Com/F_InitializeCommunication.TcPOU
FUNCTION F_InitializeCommunication : BOOL
(**************************************************************************************
 * 	Application		:	BoxControl Framework
 *	Revision		:	$Revision: 404529 $
 *	Revision date	:	$Date: 2018-04-23 08:21:38 +0200 (Mo., 23 Apr 2018) $
 *	Last changed by	:	$Author: b7bolm $
 *	URL				:	$URL: http://almscdc.swisslog.com/repo/SWPD/Development/BoxControlFramework/20_Release/trunk/01_Software/BCF/BCF/JumpStart/20_Product/10_App/11_Com/10_Lib/F_InitializeCommunication.TcPOU $
 *
 *	Purpose			:	Initialize communication
 *
 * ------------------------------------------------------------------------------------
 *	Copyright Swisslog [IP AG], Switzerland. All rights reserved.
 * 
 * ------------------------------------------------------------------------------------
 *	
 * 	Revision History: 
 *
 * 	VERSION			DATE			INITIALS			DESCRIPTION
 *	0.1				01.01.2001		swl					Example
 *
 **************************************************************************************)
VAR
	eMFCS_Channel	: E_MFCS_Channel;
	MFCS_Instance	: ITF_MFCS; // Instance to compare valid interfaces
END_VAR


// Loop over all MFCS channels
FOR eMFCS_Channel := E_MFCS_Channel.BEGIN_CHANNEL + 1 TO E_MFCS_Channel.END_CHANNEL - 1 DO
	// If a valid communicaition channel is configured
	IF __QUERYINTERFACE(fbMFCS_Channel[eMFCS_Channel], MFCS_Instance) THEN
		// Initialize channel
		fbMFCS_Channel[eMFCS_Channel].M_Init(TRUE);
	END_IF
END_FOR

// Init ITC
fbITC_Manager.M_Init(TRUE);

END_FUNCTION

// ---- 20_Product/10_BCF/11_Conv/15_Subsystem/10_Helper/F_InitializeSubsystem.TcPOU
FUNCTION F_InitializeSubsystem : BOOL
(**************************************************************************************
 * 	Application		:	BoxControl Framework
 *	Revision		:	$Revision: 404529 $
 *	Revision date	:	$Date: 2018-04-23 08:21:38 +0200 (Mo., 23 Apr 2018) $
 *	Last changed by	:	$Author: b7bolm $
 *	URL				:	$URL: http://almscdc.swisslog.com/repo/SWPD/Development/BoxControlFramework/20_Release/trunk/01_Software/BCF/BCF/JumpStart/20_Product/10_App/15_Subsystem/10_Lib/10_Conv/10_Functions/F_InitializeSubsystem.TcPOU $
 *
 *	Purpose			:	Initialize subsystem
 *
 * ------------------------------------------------------------------------------------
 *	Copyright Swisslog [IP AG], Switzerland. All rights reserved.
 * 
 * ------------------------------------------------------------------------------------
 *	
 * 	Revision History: 
 *
 * 	VERSION			DATE			INITIALS			DESCRIPTION
 *	0.1				01.01.2001		swl					Example
 *
 **************************************************************************************)

// If reference is valid
IF __ISVALIDREF(SubsystemRegistry.rSubsystem) THEN
	// Initialize subsystem
	SubsystemRegistry.rSubsystem.M_InitSubsystem(TRUE);
END_IF

END_FUNCTION

// ---- 20_Product/10_BCF/11_Conv/14_Groups/10_Helper/F_InitializeAllGroups.TcPOU
FUNCTION F_InitializeAllGroups :BOOL
(**************************************************************************************
 * 	Application		:	BoxControl Framework
 *	Revision		:	$Revision: 404529 $
 *	Revision date	:	$Date: 2018-04-23 08:21:38 +0200 (Mo., 23 Apr 2018) $
 *	Last changed by	:	$Author: b7bolm $
 *	URL				:	$URL: http://almscdc.swisslog.com/repo/SWPD/Development/BoxControlFramework/20_Release/trunk/01_Software/BCF/BCF/JumpStart/20_Product/10_App/14_Groups/10_Lib/10_Conv/10_Functions/F_InitializeAllGroups.TcPOU $
 *
 *	Purpose			:	Initialize all groups
 *
 * ------------------------------------------------------------------------------------
 *	Copyright Swisslog [IP AG], Switzerland. All rights reserved.
 * 
 * ------------------------------------------------------------------------------------
 *	
 * 	Revision History: 
 *
 * 	VERSION			DATE			INITIALS			DESCRIPTION
 *	0.1				01.01.2001		swl					Example
 *
 **************************************************************************************)
VAR
	eGroupNumber		: E_GroupNumber; // Group number
END_VAR


// Loop over all elements and initialize each group 
FOR eGroupNumber := E_GroupNumber.G_BEGIN_GROUP + 1 TO E_GroupNumber.G_END_GROUP - 1 DO
	// If reference is valid
	IF __ISVALIDREF(GroupRegistry[eGroupNumber].rGroup) THEN
		// Initialize group
		GroupRegistry[eGroupNumber].rGroup.M_InitGroup(TRUE);
	END_IF
END_FOR

END_FUNCTION

// ---- 20_Product/10_BCF/11_Conv/13_Elements/10_Helper/F_InitializeAllElements.TcPOU
FUNCTION F_InitializeAllElements :BOOL
(**************************************************************************************
 * 	Application		:	BoxControl Framework
 *	Revision		:	$Revision: 404529 $
 *	Revision date	:	$Date: 2018-04-23 08:21:38 +0200 (Mo., 23 Apr 2018) $
 *	Last changed by	:	$Author: b7bolm $
 *	URL				:	$URL: http://almscdc.swisslog.com/repo/SWPD/Development/BoxControlFramework/20_Release/trunk/01_Software/BCF/BCF/JumpStart/20_Product/10_App/13_Elements/10_Lib/10_Conv/10_Functions/F_InitializeAllElements.TcPOU $
 *
 *	Purpose			:	Initialize all elements
 *
 * ------------------------------------------------------------------------------------
 *	Copyright Swisslog [IP AG], Switzerland. All rights reserved.
 * 
 * ------------------------------------------------------------------------------------
 *	
 * 	Revision History: 
 *
 * 	VERSION			DATE			INITIALS			DESCRIPTION
 *	0.1				01.01.2001		swl					Example
 *
 **************************************************************************************)
VAR
	eElementNumber		: E_ElementNumber; // Element number
END_VAR


// Loop over all elements and initialize each element 
FOR eElementNumber := E_ElementNumber.E_BEGIN_ELEMENT+ 1 TO E_ElementNumber.E_END_ELEMENT- 1 DO
	// If reference is valid
	IF __ISVALIDREF(ElementRegistry[eElementNumber].rElement) THEN
		// Initialize element
		ElementRegistry[eElementNumber].rElement.M_InitElement(TRUE);
	END_IF
END_FOR

END_FUNCTION

// ---- 20_Product/10_BCF/11_Conv/12_E_Functions/10_Helper/F_InitializeAllFunctions.TcPOU
FUNCTION F_InitializeAllFunctions :BOOL
(**************************************************************************************
 * 	Application		:	BoxControl Framework
 *	Revision		:	$Revision: 404529 $
 *	Revision date	:	$Date: 2018-04-23 08:21:38 +0200 (Mo., 23 Apr 2018) $
 *	Last changed by	:	$Author: b7bolm $
 *	URL				:	$URL: http://almscdc.swisslog.com/repo/SWPD/Development/BoxControlFramework/20_Release/trunk/01_Software/BCF/BCF/JumpStart/20_Product/10_App/12_E_Functions/10_Lib/10_Conv/10_Functions/F_InitializeAllFunctions.TcPOU $
 *
 *	Purpose			:	Initialize all functions
 *
 * ------------------------------------------------------------------------------------
 *	Copyright Swisslog [IP AG], Switzerland. All rights reserved.
 * 
 * ------------------------------------------------------------------------------------
 *	
 * 	Revision History: 
 *
 * 	VERSION			DATE			INITIALS			DESCRIPTION
 *	0.1				01.01.2001		swl					Example
 *
 **************************************************************************************)
VAR
	eFunctionNumber		: E_FunctionNumber; // Function number

END_VAR

// Loop over all elements and initialize each function 
FOR eFunctionNumber := E_FunctionNumber.F_BEGIN_FUNCTION + 1 TO E_FunctionNumber.F_END_FUNCTION - 1 DO
	// If reference is valid
	IF __ISVALIDREF(FunctionRegistry[eFunctionNumber].rFunction) THEN
		// Initialize function
		FunctionRegistry[eFunctionNumber].rFunction.M_InitFunction(TRUE);
	END_IF
END_FOR

END_FUNCTION

// ---- 20_Product/10_BCF/11_Conv/09_Emulation/MainConvEmulation.TcPOU
PROGRAM MainConvEmulation
(**************************************************************************************
 * 	Application		:	BoxControl Framework
 *	Revision		:	$Revision: 404529 $
 *	Revision date	:	$Date: 2018-04-23 08:21:38 +0200 (Mo., 23 Apr 2018) $
 *	Last changed by	:	$Author: b7bolm $
 *	URL				:	$URL: http://almscdc.swisslog.com/repo/SWPD/Development/BoxControlFramework/20_Release/trunk/01_Software/BCF/BCF/JumpStart/20_Product/11_Emu/MainConvEmulation.TcPOU $
 *
 *	Purpose			:	Main emulation program call.
 *
 * ------------------------------------------------------------------------------------
 *	Copyright Swisslog [IP AG], Switzerland. All rights reserved.
 * 
 * ------------------------------------------------------------------------------------
 *	
 * 	Revision History: 
 *
 * 	VERSION			DATE			INITIALS			DESCRIPTION
 *	0.1				01.01.2001		swl					Example
 *
 **************************************************************************************)
VAR
	Init									: BOOL := FALSE; // Emulation is initialized 
	fbDebugMsg								: FB_DebugMsg; // Debug instance
	
	fbCommunicationCompositionEmulation		: FB_CommunicationCompositionEmulation; // Instance for communication composition
	fbSubsystemCompositionEmulation			: FB_SubsystemCompositionEmulation; // Instance for group composition
	fbGroupCompositionEmulation				: FB_GroupCompositionEmulation; // Instance for group composition
	fbElementCompositionEmulation			: FB_ElementCompositionEmulation; // Instance for element composition
	fbFunctionCompositionEmulation			: FB_FunctionCompositionEmulation; // Instance for function composition
END_VAR

(**************************************************************************************************************
   Initialize program
***************************************************************************************************************)
A_Init();

(**************************************************************************************************************
   Call Emulation
***************************************************************************************************************)
// Emulation is active
EmulationActive := Init;

IF Init THEN
	// Update references
	F_UpdateReferencesEmulation();

	// Call communication
	fbCommunicationCompositionEmulation();
		
	// Call Subsystem
	fbSubsystemCompositionEmulation();
	
	// Call groups
	fbGroupCompositionEmulation();
			
	// Call elements
	fbElementCompositionEmulation();

	// Call functions
	fbFunctionCompositionEmulation();

END_IF

ACTION A_Init:
(**************************************************************************************
 * 	NAME		A_Init
 * 	FUNCTION	Initialization
 **************************************************************************************)

// Initialize emulation after main program is initialized
IF MainConv.Init AND NOT Init THEN

	// Send debug message
	fbDebugMsg.M_SendInfoMsg('Emulation Main initialized.');

	// Load emulation configuration
	F_ConfigProductEmulation();
	F_ConfigCommunicationEmulation();
	F_ConfigPositionEmulation();
	F_ConfigGroupEmulation();
	F_ConfigSubsystemEmulation();
	
	// Set emulation initialized
	Init := TRUE;
END_IF
END_ACTION

END_PROGRAM

// ---- 20_Product/10_BCF/11_Conv/10_Base/FB_CommunicationCompositionEmulation.TcPOU
FUNCTION_BLOCK FB_CommunicationCompositionEmulation
(**************************************************************************************
 * 	Application		:	BoxControl Framework
 *	Revision		:	$Revision: 404529 $
 *	Revision date	:	$Date: 2018-04-23 08:21:38 +0200 (Mo., 23 Apr 2018) $
 *	Last changed by	:	$Author: b7bolm $
 *	URL				:	$URL: http://almscdc.swisslog.com/repo/SWPD/Development/BoxControlFramework/20_Release/trunk/01_Software/BCF/BCF/JumpStart/20_Product/11_Emu/10_Base/10_Lib/10_Conv/FB_CommunicationCompositionEmulation.TcPOU $
 *
 *	Purpose			:	Communication emulation program call.
 *
 * ------------------------------------------------------------------------------------
 *	Copyright Swisslog [IP AG], Switzerland. All rights reserved.
 * 
 * ------------------------------------------------------------------------------------
 *	
 * 	Revision History: 
 *
 * 	VERSION			DATE			INITIALS			DESCRIPTION
 *	0.1				01.01.2001		swl					Example
 *
 **************************************************************************************)
VAR
	eMFCS_Channel				: E_MFCS_Channel; // Iterator MFCS channel
	MFCS_Emulation_Instance		: ITF_MFCS_Emulation; // Instance to compare valid interfaces
	MFCS_Instance				: ITF_MFCS; // Instance to compare valid interfaces
END_VAR



(**************************************************************************************************************
   Call emulation handler for each MFCS channel
***************************************************************************************************************)
//Call all channels
FOR eMFCS_Channel := E_MFCS_Channel.BEGIN_CHANNEL + 1 TO E_MFCS_Channel.END_CHANNEL - 1 DO
	// Emulation channel is valid
	IF __QUERYINTERFACE(fbMFCS_ChannelEmulation[eMFCS_Channel], MFCS_Emulation_Instance) THEN
		// Real channel is valid too
		IF __QUERYINTERFACE(fbMFCS_Channel[eMFCS_Channel], MFCS_Instance) THEN
			// Call emulation
			fbMFCS_ChannelEmulation[eMFCS_Channel].M_ProcessData(
				meChannelSrc	:= eMFCS_Channel,
				mData 			:= fbMFCS_Channel[eMFCS_Channel].M_GetReceivedData());
		END_IF
	END_IF
END_FOR

END_FUNCTION_BLOCK

// ---- 20_Product/10_BCF/11_Conv/10_Base/FB_SubSystemCompositionEmulation.TcPOU
FUNCTION_BLOCK FB_SubsystemCompositionEmulation
(**************************************************************************************
 * 	Application		:	BoxControl Framework
 *	Revision		:	$Revision: 404529 $
 *	Revision date	:	$Date: 2018-04-23 08:21:38 +0200 (Mo., 23 Apr 2018) $
 *	Last changed by	:	$Author: b7bolm $
 *	URL				:	$URL: http://almscdc.swisslog.com/repo/SWPD/Development/BoxControlFramework/20_Release/trunk/01_Software/BCF/BCF/JumpStart/20_Product/11_Emu/10_Base/10_Lib/10_Conv/FB_SubSystemCompositionEmulation.TcPOU $
 *
 *	Purpose			:	Subsystem emulation program call.
 *
 * ------------------------------------------------------------------------------------
 *	Copyright Swisslog [IP AG], Switzerland. All rights reserved.
 * 
 * ------------------------------------------------------------------------------------
 *	
 * 	Revision History: 
 *
 * 	VERSION			DATE			INITIALS			DESCRIPTION
 *	0.1				01.01.2001		swl					Example
 *
 **************************************************************************************)
VAR
	rSubsystem		: REFERENCE TO FB_BaseObjectEmulation; // Reference
	fbDebugMsg			: FB_DebugMsg; // Debug Msg Manager (STACK) 
	DebugMsg			: T_MAXSTRING; // Debug msg
END_VAR


(**************************************************************************************************************
  Call Subsystem emulation
***************************************************************************************************************)

// If a valid reference is available 
IF __ISVALIDREF(SubsystemRegistryEmulation.rSubsystem) THEN
	// Call emulation subsystem 
	SubsystemRegistryEmulation.rSubsystem();

ELSE		
	// Invalid reference
	DebugMsg := 'FSubsystemCompositionEmulation - Reference not valid';
	fbDebugMsg.M_SendErrorMsg(mMessage := DebugMsg);
END_IF

END_FUNCTION_BLOCK

// ---- 20_Product/10_BCF/10_Base/FB_BaseObjectEmulation.TcPOU
FUNCTION_BLOCK FB_BaseObjectEmulation
(**************************************************************************************
 * 	Application		:	BoxControl Framework
 *	Revision		:	$Revision: 404529 $
 *	Revision date	:	$Date: 2018-04-23 08:21:38 +0200 (Mo., 23 Apr 2018) $
 *	Last changed by	:	$Author: b7bolm $
 *	URL				:	$URL: http://almscdc.swisslog.com/repo/SWPD/Development/BoxControlFramework/20_Release/trunk/01_Software/BCF/BCF/JumpStart/20_Product/11_Emu/10_Base/10_Lib/FB_BaseObjectEmulation.TcPOU $
 *
 *	Purpose			:	Base object emulation
 *
 * ------------------------------------------------------------------------------------
 *	Copyright Swisslog [IP AG], Switzerland. All rights reserved.
 * 
 * ------------------------------------------------------------------------------------
 *	
 * 	Revision History: 
 *
 * 	VERSION			DATE			INITIALS			DESCRIPTION
 *	0.1				01.01.2001		swl					Example
 *
 **************************************************************************************)
VAR
	fbDebugMsg		: FB_DebugMsg; // Debug instance
	DebugMsg		: T_MAXSTRING; // Debug msg
END_VAR

(**************************************************************************************************************
   Body never called!
***************************************************************************************************************)
;

METHOD M_ITC_ProcessMsg : BOOL
VAR_INPUT
	meChannelSrc		: E_MFCS_CHANNEL; // Number of the source 
	mMsgType			: INT; // Message type
	mpData				: PVOID; // Data  pointer 
	mLen				: UDINT; // Data length
END_VAR
(*
This method serves as dummy to fullfil interface requirements.

This is needed to keep independency between library product types.

This method should be overwriten in each Rootclass underneath.

*)
END_METHOD

END_FUNCTION_BLOCK

// ---- 20_Product/10_BCF/11_Conv/10_Base/FB_GroupCompositionEmulation.TcPOU
FUNCTION_BLOCK FB_GroupCompositionEmulation
(**************************************************************************************
 * 	Application		:	BoxControl Framework
 *	Revision		:	$Revision: 404529 $
 *	Revision date	:	$Date: 2018-04-23 08:21:38 +0200 (Mo., 23 Apr 2018) $
 *	Last changed by	:	$Author: b7bolm $
 *	URL				:	$URL: http://almscdc.swisslog.com/repo/SWPD/Development/BoxControlFramework/20_Release/trunk/01_Software/BCF/BCF/JumpStart/20_Product/11_Emu/10_Base/10_Lib/10_Conv/FB_GroupCompositionEmulation.TcPOU $
 *
 *	Purpose			:	Group emulation program call.
 *
 * ------------------------------------------------------------------------------------
 *	Copyright Swisslog [IP AG], Switzerland. All rights reserved.
 * 
 * ------------------------------------------------------------------------------------
 *	
 * 	Revision History: 
 *
 * 	VERSION			DATE			INITIALS			DESCRIPTION
 *	0.1				01.01.2001		swl					Example
 *
 **************************************************************************************)
VAR
	eGroupNumber		: E_GroupNumber; // Number of the Group 
	fbDebugMsg			: FB_DebugMsg; // Debug Msg Manager (STACK) 
	DebugMsg			: T_MAXSTRING; // Debug msg
END_VAR

(**************************************************************************************************************
  Call all emulation groups
***************************************************************************************************************)

// Loop trough all groups 
FOR eGroupNumber := G_BEGIN_GROUP + 1 TO G_END_GROUP - 1 DO
	// If the real is enabled 
	IF GroupRegistry[eGroupNumber].Enable THEN

		// If a valid reference is available 
		IF __ISVALIDREF(GroupRegistryEmulation[eGroupNumber].rGroup) THEN
			// Call emulation group 
			GroupRegistryEmulation[eGroupNumber].rGroup(eGroupNumber := eGroupNumber);
		ELSE		
			// Invalid reference
			DebugMsg := CONCAT('F_GroupCompositionEmulation - Reference not valid, Group index: ', INT_TO_STRING(eGroupNumber));
			fbDebugMsg.M_SendErrorMsg(mMessage := DebugMsg);
		END_IF
	END_IF
END_FOR

END_FUNCTION_BLOCK

// ---- 20_Product/10_BCF/11_Conv/10_Base/FB_ElementCompositionEmulation.TcPOU
FUNCTION_BLOCK FB_ElementCompositionEmulation
(**************************************************************************************
 * 	Application		:	BoxControl Framework
 *	Revision		:	$Revision: 404529 $
 *	Revision date	:	$Date: 2018-04-23 08:21:38 +0200 (Mo., 23 Apr 2018) $
 *	Last changed by	:	$Author: b7bolm $
 *	URL				:	$URL: http://almscdc.swisslog.com/repo/SWPD/Development/BoxControlFramework/20_Release/trunk/01_Software/BCF/BCF/JumpStart/20_Product/11_Emu/10_Base/10_Lib/10_Conv/FB_ElementCompositionEmulation.TcPOU $
 *
 *	Purpose			:	Element emulation program call.
 *
 * ------------------------------------------------------------------------------------
 *	Copyright Swisslog [IP AG], Switzerland. All rights reserved.
 * 
 * ------------------------------------------------------------------------------------
 *	
 * 	Revision History: 
 *
 * 	VERSION			DATE			INITIALS			DESCRIPTION
 *	0.1				01.01.2001		swl					Example
 *
 **************************************************************************************)
VAR
	eElementNumber		: E_ElementNumber; // Number of the element 
	fbDebugMsg			: FB_DebugMsg; // Debug Msg Manager (STACK) 
	DebugMsg			: T_MAXSTRING; // Debug msg
END_VAR

(**************************************************************************************************************
  Call all emulation elements
***************************************************************************************************************)

// Loop trough all elements 
FOR eElementNumber := E_BEGIN_ELEMENT + 1 TO E_END_ELEMENT - 1 DO
	// If this element is enabled 
	IF ElementRegistry[eElementNumber].Enable THEN
		// If a valid reference is available 
		IF __ISVALIDREF(ElementRegistryEmulation[eElementNumber].rElement) THEN
			// Call element 
			ElementRegistryEmulation[eElementNumber].rElement(eElementNumber := eElementNumber);
		ELSE
			// Invalid reference
			DebugMsg := CONCAT('F_ElementCompositionEmulation - Reference not valid, Element index: ', INT_TO_STRING(eElementNumber));
			fbDebugMsg.M_SendErrorMsg(mMessage := DebugMsg);
		END_IF
	END_IF
END_FOR

END_FUNCTION_BLOCK

// ---- 20_Product/10_BCF/11_Conv/10_Base/FB_FunctionCompositionEmulation.TcPOU
FUNCTION_BLOCK FB_FunctionCompositionEmulation
(**************************************************************************************
 * 	Application		:	BoxControl Framework
 *	Revision		:	$Revision: 404529 $
 *	Revision date	:	$Date: 2018-04-23 08:21:38 +0200 (Mo., 23 Apr 2018) $
 *	Last changed by	:	$Author: b7bolm $
 *	URL				:	$URL: http://almscdc.swisslog.com/repo/SWPD/Development/BoxControlFramework/20_Release/trunk/01_Software/BCF/BCF/JumpStart/20_Product/11_Emu/10_Base/10_Lib/10_Conv/FB_FunctionCompositionEmulation.TcPOU $
 *
 *	Purpose			:	Function emulation program call.
 *
 * ------------------------------------------------------------------------------------
 *	Copyright Swisslog [IP AG], Switzerland. All rights reserved.
 * 
 * ------------------------------------------------------------------------------------
 *	
 * 	Revision History: 
 *
 * 	VERSION			DATE			INITIALS			DESCRIPTION
 *	0.1				01.01.2001		swl					Example
 *
 **************************************************************************************)
VAR
	eFunctionNumber		: E_FunctionNumber; // Number of the function 
	fbDebugMsg			: FB_DebugMsg; // Debug Msg Manager (STACK) 
	DebugMsg			: T_MAXSTRING; // Debug msg
END_VAR

(**************************************************************************************************************
  Call all emulation functions
***************************************************************************************************************)

// Loop trough all functions 
FOR eFunctionNumber := E_FunctionNumber.F_BEGIN_FUNCTION + 1 TO E_FunctionNumber.F_END_FUNCTION - 1 DO
	// If this function is enabled 
	IF FunctionRegistry[eFunctionNumber].Enable THEN
		// If a valid reference is available 
		IF __ISVALIDREF(FunctionRegistryEmulation[eFunctionNumber].rFunction) THEN
			// Call function 
			FunctionRegistryEmulation[eFunctionNumber].rFunction(eFunctionNumber := eFunctionNumber);
		ELSE
			// Invalid reference
			DebugMsg := CONCAT('F_FunctionCompositionEmulation - Reference not valid, Function index: ', INT_TO_STRING(eFunctionNumber));
			fbDebugMsg.M_SendErrorMsg(mMessage := DebugMsg);
		END_IF
	END_IF
END_FOR

END_FUNCTION_BLOCK

// ---- 10_Project/11_Emu/10_Config/F_UpdateReferencesEmulation.TcPOU
FUNCTION F_UpdateReferencesEmulation



SubsystemRegistryEmulation.rSubsystem                                      REF= fbSubsystem10_Emulation;
GroupRegistryEmulation[E_GroupNumber.G_SG_001].rGroup                      REF= fbSG_001_Emulation;
ElementRegistryEmulation[E_ElementNumber.E_10_001_0200_00_0].rElement      REF= fbEL_10_001_0200_00_0_Emulation;
FunctionRegistryEmulation[E_FunctionNumber.F_10_001_0200_01_0].rFunction   REF= fbF_10_001_0200_01_0_Emulation;
FunctionRegistryEmulation[E_FunctionNumber.F_10_001_0200_02_0].rFunction   REF= fbF_10_001_0200_02_0_Emulation;
ElementRegistryEmulation[E_ElementNumber.E_10_001_0201_00_0].rElement      REF= fbEL_10_001_0201_00_0_Emulation;
FunctionRegistryEmulation[E_FunctionNumber.F_10_001_0201_01_0].rFunction   REF= fbF_10_001_0201_01_0_Emulation;
ElementRegistryEmulation[E_ElementNumber.E_10_001_0202_00_0].rElement      REF= fbEL_10_001_0202_00_0_Emulation;
FunctionRegistryEmulation[E_FunctionNumber.F_10_001_0202_01_0].rFunction   REF= fbF_10_001_0202_01_0_Emulation;
ElementRegistryEmulation[E_ElementNumber.E_10_001_0203_00_0].rElement      REF= fbEL_10_001_0203_00_0_Emulation;
FunctionRegistryEmulation[E_FunctionNumber.F_10_001_0203_01_0].rFunction   REF= fbF_10_001_0203_01_0_Emulation;
FunctionRegistryEmulation[E_FunctionNumber.F_10_001_0203_02_0].rFunction   REF= fbF_10_001_0203_02_0_Emulation;
FunctionRegistryEmulation[E_FunctionNumber.F_10_001_0203_03_0].rFunction   REF= fbF_10_001_0203_03_0_Emulation;
FunctionRegistryEmulation[E_FunctionNumber.F_10_001_0203_04_0].rFunction   REF= fbF_10_001_0203_04_0_Emulation;
FunctionRegistryEmulation[E_FunctionNumber.F_10_001_0203_05_0].rFunction   REF= fbF_10_001_0203_05_0_Emulation;
ElementRegistryEmulation[E_ElementNumber.E_10_001_0204_00_0].rElement      REF= fbEL_10_001_0204_00_0_Emulation;
FunctionRegistryEmulation[E_FunctionNumber.F_10_001_0204_01_0].rFunction   REF= fbF_10_001_0204_01_0_Emulation;
ElementRegistryEmulation[E_ElementNumber.E_10_001_0205_00_0].rElement      REF= fbEL_10_001_0205_00_0_Emulation;
ElementRegistryEmulation[E_ElementNumber.E_10_001_0207_00_0].rElement      REF= fbEL_10_001_0207_00_0_Emulation;
FunctionRegistryEmulation[E_FunctionNumber.F_10_001_0207_01_0].rFunction   REF= fbF_10_001_0207_01_0_Emulation;
FunctionRegistryEmulation[E_FunctionNumber.F_10_001_0207_02_0].rFunction   REF= fbF_10_001_0207_02_0_Emulation;
ElementRegistryEmulation[E_ElementNumber.E_10_001_0208_00_0].rElement      REF= fbEL_10_001_0208_00_0_Emulation;
FunctionRegistryEmulation[E_FunctionNumber.F_10_001_0208_01_0].rFunction   REF= fbF_10_001_0208_01_0_Emulation;
ElementRegistryEmulation[E_ElementNumber.E_10_001_0209_00_0].rElement      REF= fbEL_10_001_0209_00_0_Emulation;
FunctionRegistryEmulation[E_FunctionNumber.F_10_001_0209_01_0].rFunction   REF= fbF_10_001_0209_01_0_Emulation;
ElementRegistryEmulation[E_ElementNumber.E_10_001_0211_00_0].rElement      REF= fbEL_10_001_0211_00_0_Emulation;
FunctionRegistryEmulation[E_FunctionNumber.F_10_001_0211_01_0].rFunction   REF= fbF_10_001_0211_01_0_Emulation;
ElementRegistryEmulation[E_ElementNumber.E_10_001_0212_00_0].rElement      REF= fbEL_10_001_0212_00_0_Emulation;
FunctionRegistryEmulation[E_FunctionNumber.F_10_001_0212_01_0].rFunction   REF= fbF_10_001_0212_01_0_Emulation;
ElementRegistryEmulation[E_ElementNumber.E_10_001_0213_00_0].rElement      REF= fbEL_10_001_0213_00_0_Emulation;
FunctionRegistryEmulation[E_FunctionNumber.F_10_001_0213_01_0].rFunction   REF= fbF_10_001_0213_01_0_Emulation;
FunctionRegistryEmulation[E_FunctionNumber.F_10_001_0213_02_0].rFunction   REF= fbF_10_001_0213_02_0_Emulation;
ElementRegistryEmulation[E_ElementNumber.E_10_001_0214_00_0].rElement      REF= fbEL_10_001_0214_00_0_Emulation;
FunctionRegistryEmulation[E_FunctionNumber.F_10_001_0214_01_0].rFunction   REF= fbF_10_001_0214_01_0_Emulation;
ElementRegistryEmulation[E_ElementNumber.E_10_001_0215_00_0].rElement      REF= fbEL_10_001_0215_00_0_Emulation;
FunctionRegistryEmulation[E_FunctionNumber.F_10_001_0215_01_0].rFunction   REF= fbF_10_001_0215_01_0_Emulation;
FunctionRegistryEmulation[E_FunctionNumber.F_10_001_0215_02_0].rFunction   REF= fbF_10_001_0215_02_0_Emulation;
FunctionRegistryEmulation[E_FunctionNumber.F_10_001_0215_03_0].rFunction   REF= fbF_10_001_0215_03_0_Emulation;
ElementRegistryEmulation[E_ElementNumber.E_10_001_0216_00_0].rElement      REF= fbEL_10_001_0216_00_0_Emulation;
FunctionRegistryEmulation[E_FunctionNumber.F_10_001_0216_01_0].rFunction   REF= fbF_10_001_0216_01_0_Emulation;
FunctionRegistryEmulation[E_FunctionNumber.F_10_001_0216_02_0].rFunction   REF= fbF_10_001_0216_02_0_Emulation;
ElementRegistryEmulation[E_ElementNumber.E_10_001_0217_00_0].rElement      REF= fbEL_10_001_0217_00_0_Emulation;
FunctionRegistryEmulation[E_FunctionNumber.F_10_001_0217_01_0].rFunction   REF= fbF_10_001_0217_01_0_Emulation;
ElementRegistryEmulation[E_ElementNumber.E_10_001_0218_00_0].rElement      REF= fbEL_10_001_0218_00_0_Emulation;
FunctionRegistryEmulation[E_FunctionNumber.F_10_001_0218_01_0].rFunction   REF= fbF_10_001_0218_01_0_Emulation;
ElementRegistryEmulation[E_ElementNumber.E_10_001_0219_00_0].rElement      REF= fbEL_10_001_0219_00_0_Emulation;
FunctionRegistryEmulation[E_FunctionNumber.F_10_001_0219_01_0].rFunction   REF= fbF_10_001_0219_01_0_Emulation;
ElementRegistryEmulation[E_ElementNumber.E_10_001_0220_00_0].rElement      REF= fbEL_10_001_0220_00_0_Emulation;
FunctionRegistryEmulation[E_FunctionNumber.F_10_001_0220_01_0].rFunction   REF= fbF_10_001_0220_01_0_Emulation;
ElementRegistryEmulation[E_ElementNumber.E_10_001_0221_00_0].rElement      REF= fbEL_10_001_0221_00_0_Emulation;
FunctionRegistryEmulation[E_FunctionNumber.F_10_001_0221_01_0].rFunction   REF= fbF_10_001_0221_01_0_Emulation;
ElementRegistryEmulation[E_ElementNumber.E_10_001_0222_00_0].rElement      REF= fbEL_10_001_0222_00_0_Emulation;
FunctionRegistryEmulation[E_FunctionNumber.F_10_001_0222_01_0].rFunction   REF= fbF_10_001_0222_01_0_Emulation;
ElementRegistryEmulation[E_ElementNumber.E_10_001_0223_00_0].rElement      REF= fbEL_10_001_0223_00_0_Emulation;
ElementRegistryEmulation[E_ElementNumber.E_10_001_0225_00_0].rElement      REF= fbEL_10_001_0225_00_0_Emulation;
FunctionRegistryEmulation[E_FunctionNumber.F_10_001_0225_01_0].rFunction   REF= fbF_10_001_0225_01_0_Emulation;
ElementRegistryEmulation[E_ElementNumber.E_10_001_0226_00_0].rElement      REF= fbEL_10_001_0226_00_0_Emulation;
FunctionRegistryEmulation[E_FunctionNumber.F_10_001_0226_01_0].rFunction   REF= fbF_10_001_0226_01_0_Emulation;
ElementRegistryEmulation[E_ElementNumber.E_10_001_0227_00_0].rElement      REF= fbEL_10_001_0227_00_0_Emulation;
FunctionRegistryEmulation[E_FunctionNumber.F_10_001_0227_01_0].rFunction   REF= fbF_10_001_0227_01_0_Emulation;
ElementRegistryEmulation[E_ElementNumber.E_10_001_0230_00_0].rElement      REF= fbEL_10_001_0230_00_0_Emulation;
FunctionRegistryEmulation[E_FunctionNumber.F_10_001_0230_01_0].rFunction   REF= fbF_10_001_0230_01_0_Emulation;
ElementRegistryEmulation[E_ElementNumber.E_10_001_0232_00_0].rElement      REF= fbEL_10_001_0232_00_0_Emulation;
FunctionRegistryEmulation[E_FunctionNumber.F_10_001_0232_01_0].rFunction   REF= fbF_10_001_0232_01_0_Emulation;
FunctionRegistryEmulation[E_FunctionNumber.F_10_001_0232_02_0].rFunction   REF= fbF_10_001_0232_02_0_Emulation;
ElementRegistryEmulation[E_ElementNumber.E_10_001_0233_00_0].rElement      REF= fbEL_10_001_0233_00_0_Emulation;
FunctionRegistryEmulation[E_FunctionNumber.F_10_001_0233_01_0].rFunction   REF= fbF_10_001_0233_01_0_Emulation;
GroupRegistryEmulation[E_GroupNumber.G_SG_002].rGroup                      REF= fbSG_002_Emulation;
ElementRegistryEmulation[E_ElementNumber.E_10_002_0206_00_0].rElement      REF= fbEL_10_002_0206_00_0_Emulation;
FunctionRegistryEmulation[E_FunctionNumber.F_10_002_0206_01_0].rFunction   REF= fbF_10_002_0206_01_0_Emulation;

END_FUNCTION

// ---- 10_Project/11_Emu/10_Config/F_ConfigProductEmulation.TcPOU
FUNCTION F_ConfigProductEmulation : BOOL



(****************************************************************************************
   Configuration Product
*****************************************************************************************)
fbITC_ManagerEmulation := fbITC_ConveyorEmulation;

(****************************************************************************************
   Define MFCS channels (e.g.SIS channels)
*****************************************************************************************)
fbMFCS_ChannelEmulation[E_MFCS_Channel.AM] 		:= fbMFCS_SIS_AM_Emulation;
fbMFCS_ChannelEmulation[E_MFCS_Channel.SPOC]	:= fbMFCS_SIS_SPOC_Emulation;
fbMFCS_ChannelEmulation[E_MFCS_Channel.LOGGING] := fbMFCS_SIS_LOG_Emulation;

END_FUNCTION

// ---- 10_Project/11_Emu/10_Config/F_ConfigCommunicationEmulation.TcPOU
FUNCTION F_ConfigCommunicationEmulation : BOOL

;

END_FUNCTION

// ---- 10_Project/11_Emu/10_Config/F_ConfigPositionEmulation.TcPOU
FUNCTION F_ConfigPositionEmulation



F_ConfigPositionEmulation_001();

